KUKA KRL program: MyProgram_090().src

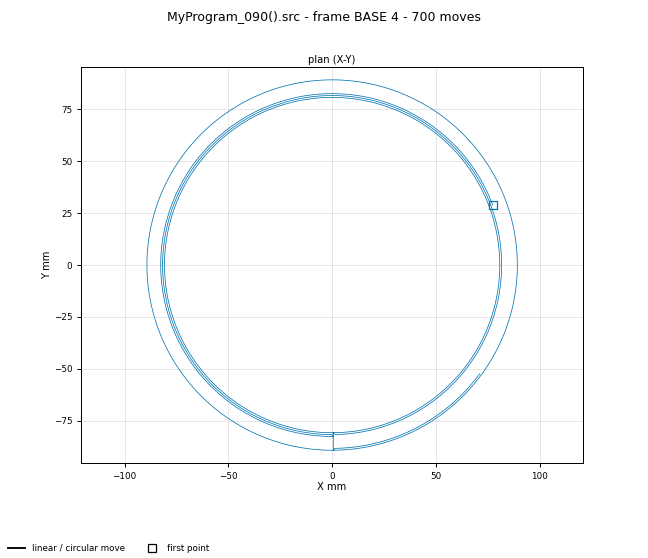
[picture p0: tool path of MyProgram_090().src in frame BASE 4, 700 of 700 moves have a stored position in this frame; points joined in program order, loops and branches not executed]
&ACCESS RVP
&REL 1
&PARAM TEMPLATE = C:\KRC\Roboter\Template\vorgabe
&PARAM EDITMASK = *
DEF MyProgram_090()
; ---- Setting reference (Base) ----
$BASE = BASE_DATA[4]

; --------------------------
; ---- Setting tool (TCP) ----
$TOOL = TOOL_DATA[3]
; --------------------------

$VEL.CP = VEL_APROX_PRINT
Startdeposition()
$VEL.CP = VEL_PRINT
LIN {X 77.3281,Y 28.9448,Z 86,A 15.3349,B 24.9023,C -2.2824,E1 25.1495,E2 429.3591} C_DIS
LIN {X 75.8466,Y 32.631,Z 86,A 18.4549,B 24.9006,C -2.3023,E1 25.1461,E2 426.2095} C_DIS
LIN {X 74.568,Y 35.455,Z 86,A 20.5991,B 24.9001,C -2.3081,E1 25.1436,E2 424.0632} C_DIS
LIN {X 72.599,Y 39.3284,Z 86,A 23.5098,B 24.8996,C -2.3129,E1 25.1398,E2 421.1565} C_DIS
LIN {X 70.8215,Y 42.4488,Z 86,A 26.772,B 24.8968,C -2.3448,E1 25.1351,E2 417.8357} C_DIS
LIN {X 68.6878,Y 45.8205,Z 86,A 28.6373,B 24.8988,C -2.3222,E1 25.1323,E2 416.0329} C_DIS
LIN {X 67.0803,Y 48.1416,Z 86,A 30.6371,B 24.8983,C -2.3285,E1 25.1291,E2 414.0282} C_DIS
LIN {X 63.6188,Y 52.6309,Z 86,A 34.2149,B 24.8985,C -2.3263,E1 25.123,E2 410.4722} C_DIS
LIN {X 61.7276,Y 54.8374,Z 86,A 37.2047,B 24.8953,C -2.3623,E1 25.1174,E2 407.4109} C_DIS
LIN {X 59.4279,Y 57.3206,Z 86,A 39.1109,B 24.8961,C -2.3531,E1 25.1137,E2 405.5347} C_DIS
LIN {X 57.4607,Y 59.2929,Z 86,A 40.8256,B 24.8964,C -2.3501,E1 25.1103,E2 403.8342} C_DIS
LIN {X 55.1536,Y 61.4445,Z 86,A 43.0458,B 24.8959,C -2.3555,E1 25.1058,E2 401.6102} C_DIS
LIN {X 52.6987,Y 63.5625,Z 86,A 45.3521,B 24.8953,C -2.3616,E1 25.1008,E2 399.2985} C_DIS
LIN {X 48.15,Y 67.0743,Z 86,A 49.5371,B 24.8942,C -2.3748,E1 25.0915,E2 395.0973} C_DIS
LIN {X 45.0145,Y 69.219,Z 86,A 51.9336,B 24.8945,C -2.3714,E1 25.0859,E2 392.7168} C_DIS
LIN {X 39.6414,Y 72.4292,Z 86,A 55.9168,B 24.8949,C -2.3664,E1 25.0764,E2 388.7575} C_DIS
LIN {X 35.4802,Y 74.5559,Z 86,A 59.3138,B 24.8941,C -2.3753,E1 25.0679,E2 385.3489} C_DIS
LIN {X 32.5804,Y 75.8687,Z 86,A 61.5876,B 24.8937,C -2.3797,E1 25.0621,E2 383.0701} C_DIS
LIN {X 30.2189,Y 76.8385,Z 86,A 63.6936,B 24.8926,C -2.3918,E1 25.0565,E2 380.9401} C_DIS
LIN {X 26.6751,Y 78.14,Z 86,A 66.6036,B 24.8916,C -2.403,E1 25.0488,E2 378.0094} C_DIS
LIN {X 23.5557,Y 79.1357,Z 86,A 67.8541,B 24.8943,C -2.3735,E1 25.0457,E2 376.8311} C_DIS
LIN {X 20.2883,Y 80.0362,Z 86,A 70.6318,B 24.893,C -2.3879,E1 25.0381,E2 374.0238} C_DIS
LIN {X 17.3744,Y 80.7187,Z 86,A 72.792,B 24.8927,C -2.3915,E1 25.0322,E2 371.858} C_DIS
LIN {X 14.1692,Y 81.3435,Z 86,A 75.1053,B 24.8925,C -2.3937,E1 25.0258,E2 369.5418} C_DIS
LIN {X 11.6124,Y 81.7465,Z 86,A 77.0151,B 24.8921,C -2.3976,E1 25.0205,E2 367.6245} C_DIS
LIN {X 8.7977,Y 82.0973,Z 86,A 78.7957,B 24.8926,C -2.3923,E1 25.0156,E2 365.8578} C_DIS
LIN {X 5.8329,Y 82.3613,Z 86,A 80.8527,B 24.8926,C -2.3922,E1 25.0099,E2 363.8021} C_DIS
LIN {X 2.46,Y 82.5305,Z 86,A 83.3881,B 24.8921,C -2.3977,E1 25.0028,E2 361.2543} C_DIS
LIN {X -1.694,Y 82.5499,Z 86,A 85.9176,B 24.8931,C -2.3867,E1 24.9958,E2 358.751} C_DIS
LIN {X -4.2402,Y 82.4588,Z 86,A 87.9133,B 24.8926,C -2.3927,E1 24.9902,E2 356.7404} C_DIS
LIN {X -7.701,Y 82.2073,Z 86,A 90.4483,B 24.8923,C -2.3954,E1 24.9831,E2 354.198} C_DIS
LIN {X -11.3944,Y 81.7774,Z 86,A 92.4535,B 24.894,C -2.3771,E1 24.9777,E2 352.2347} C_DIS
LIN {X -13.5496,Y 81.4478,Z 86,A 94.2689,B 24.8933,C -2.3848,E1 24.9726,E2 350.3994} C_DIS
LIN {X -16.7265,Y 80.8552,Z 86,A 97.0733,B 24.892,C -2.3992,E1 24.9649,E2 347.5575} C_DIS
LIN {X -20.9138,Y 79.8754,Z 86,A 100.2073,B 24.8918,C -2.4006,E1 24.9564,E2 344.4156} C_DIS
LIN {X -24.2643,Y 78.9213,Z 86,A 102.3651,B 24.8928,C -2.3905,E1 24.9506,E2 342.2784} C_DIS
LIN {X -27.4735,Y 77.8624,Z 86,A 105.2276,B 24.8917,C -2.4024,E1 24.943,E2 339.3818} C_DIS
LIN {X -31.5003,Y 76.3231,Z 86,A 107.3625,B 24.8943,C -2.3738,E1 24.9377,E2 337.3103} C_DIS
LIN {X -34.3091,Y 75.1026,Z 86,A 109.4716,B 24.8946,C -2.3702,E1 24.9323,E2 335.2046} C_DIS
LIN {X -37.1656,Y 73.731,Z 86,A 112.4576,B 24.8929,C -2.3889,E1 24.9247,E2 332.1661} C_DIS
LIN {X -40.6338,Y 71.8778,Z 86,A 114.2221,B 24.8957,C -2.3572,E1 24.9206,E2 330.4722} C_DIS
LIN {X -43.0737,Y 70.4418,Z 86,A 116.6537,B 24.8949,C -2.3666,E1 24.9147,E2 328.0106} C_DIS
LIN {X -46.8346,Y 67.9989,Z 86,A 119.7688,B 24.8954,C -2.3607,E1 24.9075,E2 324.8994} C_DIS
LIN {X -49.3306,Y 66.2113,Z 86,A 121.5161,B 24.8968,C -2.3457,E1 24.9036,E2 323.1816} C_DIS
LIN {X -51.6187,Y 64.4443,Z 86,A 123.7673,B 24.8965,C -2.3482,E1 24.8986,E2 320.9162} C_DIS
LIN {X -53.4699,Y 62.9151,Z 86,A 125.3426,B 24.8971,C -2.342,E1 24.8953,E2 319.3495} C_DIS
LIN {X -55.9727,Y 60.6995,Z 86,A 127.7309,B 24.8974,C -2.3386,E1 24.8903,E2 316.9597} C_DIS
LIN {X -58.3701,Y 58.3994,Z 86,A 130.1929,B 24.8974,C -2.3374,E1 24.8854,E2 314.4903} C_DIS
LIN {X -60.9993,Y 55.646,Z 86,A 132.5499,B 24.8987,C -2.3232,E1 24.881,E2 312.157} C_DIS
LIN {X -63.0145,Y 53.3532,Z 86,A 134.8528,B 24.8987,C -2.3228,E1 24.8767,E2 309.8445} C_DIS
LIN {X -65.1441,Y 50.7324,Z 86,A 137.6368,B 24.8983,C -2.3286,E1 24.8719,E2 307.0336} C_DIS
LIN {X -68.1053,Y 46.6821,Z 86,A 140.6854,B 24.9001,C -2.3074,E1 24.867,E2 304.0206} C_DIS
LIN {X -70.4763,Y 43.0168,Z 86,A 143.9951,B 24.9001,C -2.3064,E1 24.8621,E2 300.6963} C_DIS
LIN {X -72.2097,Y 40.0393,Z 86,A 146.2197,B 24.9012,C -2.2951,E1 24.859,E2 298.4871} C_DIS
LIN {X -74.9102,Y 34.7247,Z 86,A 150.4078,B 24.9021,C -2.2842,E1 24.8539,E2 294.3024} C_DIS
LIN {X -75.9626,Y 32.3591,Z 86,A 152.1687,B 24.9027,C -2.2779,E1 24.8519,E2 292.547} C_DIS
LIN {X -77.3859,Y 28.792,Z 86,A 155.1139,B 24.9027,C -2.2772,E1 24.849,E2 289.5867} C_DIS
LIN {X -78.3928,Y 25.9256,Z 86,A 156.9348,B 24.9039,C -2.263,E1 24.8474,E2 287.7893} C_DIS
LIN {X -79.896,Y 20.8338,Z 86,A 160.5723,B 24.905,C -2.2503,E1 24.8446,E2 284.1612} C_DIS
LIN {X -80.5932,Y 17.9499,Z 86,A 162.7179,B 24.9054,C -2.2461,E1 24.8433,E2 282.0131} C_DIS
LIN {X -81.3182,Y 14.3103,Z 86,A 166.0647,B 24.9043,C -2.2586,E1 24.8416,E2 278.6166} C_DIS
LIN {X -81.9179,Y 10.3374,Z 86,A 168.0108,B 24.907,C -2.2272,E1 24.8409,E2 276.7338} C_DIS
LIN {X -82.1781,Y 8.0167,Z 86,A 169.7244,B 24.9072,C -2.2245,E1 24.8404,E2 275.0165} C_DIS
LIN {X -82.4608,Y 4.2037,Z 86,A 172.2617,B 24.9081,C -2.2129,E1 24.8399,E2 272.4915} C_DIS
LIN {X -82.5537,Y 1.4888,Z 86,A 174.2134,B 24.9085,C -2.2087,E1 24.8398,E2 270.5382} C_DIS
LIN {X -82.5438,Y -2.0277,Z 86,A 176.555,B 24.9094,C -2.1983,E1 24.8398,E2 268.2073} C_DIS
LIN {X -82.4146,Y -5.0392,Z 86,A 178.8476,B 24.9094,C -2.197,E1 24.8402,E2 265.904} C_DIS
LIN {X -82.1848,Y -7.9446,Z 86,A -178.3575,B 24.9083,C -2.2113,E1 24.841,E2 263.0581} C_DIS
LIN {X -81.7181,Y -11.8118,Z 86,A -176.4955,B 24.9108,C -2.1803,E1 24.8416,E2 261.2591} C_DIS
LIN {X -80.6837,Y -17.5348,Z 86,A -172.3512,B 24.9116,C -2.1706,E1 24.8438,E2 257.1132} C_DIS
LIN {X -79.8963,Y -20.8325,Z 86,A -170.024,B 24.9123,C -2.1628,E1 24.8454,E2 254.7912} C_DIS
LIN {X -79.3316,Y -22.8909,Z 86,A -167.3362,B 24.91,C -2.191,E1 24.8476,E2 252.0204} C_DIS
LIN {X -77.7775,Y -27.7156,Z 86,A -164.7586,B 24.9129,C -2.1551,E1 24.8498,E2 249.514} C_DIS
LIN {X -76.5697,Y -30.8945,Z 86,A -162.5845,B 24.9138,C -2.1432,E1 24.852,E2 247.3559} C_DIS
LIN {X -75.4207,Y -33.6031,Z 86,A -160.5049,B 24.9142,C -2.1385,E1 24.8544,E2 245.2763} C_DIS
LIN {X -74.1285,Y -36.365,Z 86,A -158.3588,B 24.9146,C -2.1334,E1 24.857,E2 243.1307} C_DIS
LIN {X -72.0249,Y -40.3702,Z 86,A -155.0625,B 24.915,C -2.1292,E1 24.8613,E2 239.8269} C_DIS
LIN {X -69.3806,Y -44.7627,Z 86,A -151.6258,B 24.916,C -2.1166,E1 24.8664,E2 236.4027} C_DIS
LIN {X -67.4996,Y -47.554,Z 86,A -148.4036,B 24.9145,C -2.1353,E1 24.8716,E2 233.1201} C_DIS
LIN {X -64.8603,Y -51.0929,Z 86,A -146.635,B 24.9179,C -2.0922,E1 24.8745,E2 231.4459} C_DIS
LIN {X -62.2386,Y -54.2559,Z 86,A -142.7938,B 24.9163,C -2.113,E1 24.8815,E2 227.5374} C_DIS
LIN {X -60.0446,Y -56.6746,Z 86,A -141.2475,B 24.9182,C -2.088,E1 24.8844,E2 226.044} C_DIS
LIN {X -58.2822,Y -58.4863,Z 86,A -139.2971,B 24.9182,C -2.0898,E1 24.8882,E2 224.0811} C_DIS
LIN {X -54.727,Y -61.8264,Z 86,A -136.136,B 24.9191,C -2.0767,E1 24.8947,E2 220.9383} C_DIS
LIN {X -51.2494,Y -64.7367,Z 86,A -132.4233,B 24.9183,C -2.0868,E1 24.9028,E2 217.1874} C_DIS
LIN {X -47.5417,Y -67.5083,Z 86,A -129.4906,B 24.9194,C -2.0734,E1 24.9093,E2 214.2764} C_DIS
LIN {X -45.2055,Y -69.0932,Z 86,A -127.0426,B 24.9185,C -2.0844,E1 24.9151,E2 211.7943} C_DIS
LIN {X -41.413,Y -71.431,Z 86,A -124.0005,B 24.919,C -2.0785,E1 24.9224,E2 208.7569} C_DIS
LIN {X -37.1468,Y -73.7406,Z 86,A -120.9339,B 24.92,C -2.0655,E1 24.93,E2 205.7128} C_DIS
LIN {X -34.1894,Y -75.1565,Z 86,A -118.8468,B 24.9206,C -2.0575,E1 24.9352,E2 203.6396} C_DIS
LIN {X -30.8787,Y -76.5762,Z 86,A -116.3984,B 24.9209,C -2.0534,E1 24.9415,E2 201.1952} C_DIS
LIN {X -26.6206,Y -78.1584,Z 86,A -113.4742,B 24.9217,C -2.044,E1 24.9492,E2 198.2876} C_DIS
LIN {X -24.1171,Y -78.9672,Z 86,A -111.2313,B 24.9208,C -2.0549,E1 24.9552,E2 196.0149} C_DIS
LIN {X -20.8123,Y -79.9015,Z 86,A -108.9288,B 24.9211,C -2.051,E1 24.9614,E2 193.718} C_DIS
LIN {X -17.7972,Y -80.6265,Z 86,A -106.6486,B 24.9209,C -2.0538,E1 24.9676,E2 191.4283} C_DIS
LIN {X -14.6611,Y -81.2551,Z 86,A -104.2027,B 24.9204,C -2.0597,E1 24.9744,E2 188.9656} C_DIS
LIN {X -10.524,Y -81.8937,Z 86,A -101.6715,B 24.9214,C -2.0479,E1 24.9813,E2 186.4605} C_DIS
LIN {X -7.454,Y -82.2301,Z 86,A -99.5955,B 24.9215,C -2.0457,E1 24.9871,E2 184.3887} C_DIS
LIN {X -3.4693,Y -82.4943,Z 86,A -96.4906,B 24.9207,C -2.0559,E1 24.9958,E2 181.2585} C_DIS
LIN {X 0.5302,Y -82.5625,Z 86,A -94.6776,B 24.9229,C -2.0274,E1 25.0007,E2 179.5132} C_DIS
Enddeposition()
LIN {X 0.5302,Y -82.5625,Z 86,A -94.6776,B 24.9229,C -2.0274,E1 25.0007,E2 179.5132} C_DIS
Startdeposition()
$VEL.CP = VEL_PRINT
LIN {X -0.0163,Y -81.6615,Z 86,A -95.4197,B 24.9225,C -2.0324,E1 24.9986,E2 180.2432} C_DIS
LIN {X -2.7317,Y -81.6147,Z 86,A -97.1926,B 24.9223,C -2.0361,E1 24.9937,E2 182.0077} C_DIS
LIN {X -5.5212,Y -81.4732,Z 86,A -99.1546,B 24.9223,C -2.0359,E1 24.9882,E2 183.9707} C_DIS
LIN {X -8.4748,Y -81.2191,Z 86,A -101.2543,B 24.9223,C -2.0355,E1 24.9824,E2 186.0724} C_DIS
LIN {X -11.4403,Y -80.8547,Z 86,A -103.348,B 24.9223,C -2.036,E1 24.9766,E2 188.1666} C_DIS
LIN {X -14.2538,Y -80.4067,Z 86,A -105.405,B 24.9223,C -2.0349,E1 24.9709,E2 190.2281} C_DIS
LIN {X -17.4514,Y -79.7735,Z 86,A -107.7669,B 24.9224,C -2.0337,E1 24.9644,E2 192.5956} C_DIS
LIN {X -20.8127,Y -78.9648,Z 86,A -110.2307,B 24.9224,C -2.034,E1 24.9578,E2 195.0624} C_DIS
LIN {X -24.2019,Y -77.9912,Z 86,A -112.6185,B 24.9221,C -2.0382,E1 24.9514,E2 197.4442} C_DIS
LIN {X -27.44,Y -76.9129,Z 86,A -115.1204,B 24.9221,C -2.0371,E1 24.9448,E2 199.9535} C_DIS
LIN {X -30.5238,Y -75.7413,Z 86,A -117.3329,B 24.9218,C -2.0422,E1 24.939,E2 202.1586} C_DIS
LIN {X -33.4971,Y -74.4736,Z 86,A -119.5845,B 24.9216,C -2.0451,E1 24.9333,E2 204.4086} C_DIS
LIN {X -36.4481,Y -73.0749,Z 86,A -121.9228,B 24.9215,C -2.0465,E1 24.9274,E2 206.7497} C_DIS
LIN {X -39.2907,Y -71.5875,Z 86,A -124.3132,B 24.9215,C -2.0455,E1 24.9215,E2 209.149} C_DIS
LIN {X -41.5941,Y -70.273,Z 86,A -126.0513,B 24.9211,C -2.0516,E1 24.9173,E2 210.878} C_DIS
LIN {X -44.204,Y -68.6613,Z 86,A -128.0921,B 24.9206,C -2.0579,E1 24.9125,E2 212.9102} C_DIS
LIN {X -46.6315,Y -67.0363,Z 86,A -130.1603,B 24.9204,C -2.0607,E1 24.9077,E2 214.9787} C_DIS
LIN {X -49.0247,Y -65.3066,Z 86,A -133.1291,B 24.922,C -2.0399,E1 24.901,E2 218.0076} C_DIS
LIN {X -52.1622,Y -62.8289,Z 86,A -135.0796,B 24.9198,C -2.0681,E1 24.8969,E2 219.8982} C_DIS
LIN {X -54.3609,Y -60.9367,Z 86,A -137.5367,B 24.9204,C -2.0607,E1 24.8917,E2 222.3827} C_DIS
LIN {X -57.3481,Y -58.134,Z 86,A -140.1183,B 24.9193,C -2.0744,E1 24.8865,E2 224.9423} C_DIS
LIN {X -59.4283,Y -56.0058,Z 86,A -142.8327,B 24.9203,C -2.0622,E1 24.8812,E2 227.6976} C_DIS
LIN {X -61.8542,Y -53.3164,Z 86,A -144.7929,B 24.9186,C -2.0834,E1 24.8777,E2 229.6163} C_DIS
LIN {X -64.183,Y -50.487,Z 86,A -147.1554,B 24.9177,C -2.095,E1 24.8736,E2 231.9621} C_DIS
LIN {X -66.2039,Y -47.8082,Z 86,A -149.7166,B 24.9177,C -2.0952,E1 24.8693,E2 234.5351} C_DIS
LIN {X -68.0014,Y -45.2136,Z 86,A -151.9136,B 24.9172,C -2.1012,E1 24.8659,E2 236.7287} C_DIS
LIN {X -69.6279,Y -42.6663,Z 86,A -154.3798,B 24.9175,C -2.0976,E1 24.8622,E2 239.2161} C_DIS
LIN {X -72.238,Y -38.0794,Z 86,A -157.7911,B 24.9161,C -2.1152,E1 24.8576,E2 242.6033} C_DIS
LIN {X -73.688,Y -35.192,Z 86,A -160.1175,B 24.9157,C -2.1199,E1 24.8548,E2 244.931} C_DIS
LIN {X -75.1122,Y -32.0414,Z 86,A -162.5168,B 24.9151,C -2.1275,E1 24.8521,E2 247.3255} C_DIS
LIN {X -76.3612,Y -28.9367,Z 86,A -164.8125,B 24.9145,C -2.1357,E1 24.8497,E2 249.6145} C_DIS
LIN {X -77.739,Y -25.0006,Z 86,A -167.7777,B 24.9138,C -2.1433,E1 24.8471,E2 252.5785} C_DIS
LIN {X -78.6619,Y -21.927,Z 86,A -169.7895,B 24.9128,C -2.1562,E1 24.8455,E2 254.571} C_DIS
LIN {X -79.5463,Y -18.4598,Z 86,A -172.518,B 24.9126,C -2.1582,E1 24.8437,E2 257.3107} C_DIS
LIN {X -80.6981,Y -12.4973,Z 86,A -177.8758,B 24.9138,C -2.1435,E1 24.8411,E2 262.7355} C_DIS
LIN {X -81.2753,Y -7.9295,Z 86,A 179.9404,B 24.9108,C -2.1802,E1 24.8404,E2 264.8446} C_DIS
LIN {X -81.4834,Y -5.3695,Z 86,A 178.0036,B 24.9107,C -2.1825,E1 24.84,E2 266.7876} C_DIS
LIN {X -81.6368,Y -2.0114,Z 86,A 175.5316,B 24.9103,C -2.1871,E1 24.8398,E2 269.2636} C_DIS
LIN {X -81.6507,Y 1.2603,Z 86,A 173.367,B 24.9094,C -2.1977,E1 24.8398,E2 271.4157} C_DIS
LIN {X -81.5318,Y 4.5754,Z 86,A 170.3679,B 24.9102,C -2.1881,E1 24.8403,E2 274.4559} C_DIS
LIN {X -81.2554,Y 8.1284,Z 86,A 168.4292,B 24.9084,C -2.2103,E1 24.8408,E2 276.3532} C_DIS
LIN {X -80.6413,Y 12.8647,Z 86,A 165.1268,B 24.9074,C -2.2222,E1 24.842,E2 279.6469} C_DIS
LIN {X -80.1601,Y 15.5802,Z 86,A 163.3021,B 24.9066,C -2.2312,E1 24.843,E2 281.4609} C_DIS
LIN {X -79.4501,Y 18.8757,Z 86,A 160.6417,B 24.9066,C -2.2311,E1 24.8446,E2 284.1373} C_DIS
LIN {X -78.6107,Y 22.1078,Z 86,A 158.3187,B 24.906,C -2.239,E1 24.8463,E2 286.455} C_DIS
LIN {X -77.6206,Y 25.3667,Z 86,A 156.0491,B 24.9051,C -2.2494,E1 24.8482,E2 288.7125} C_DIS
LIN {X -76.7091,Y 28.0015,Z 86,A 154.0454,B 24.9047,C -2.2542,E1 24.8501,E2 290.7162} C_DIS
LIN {X -75.5189,Y 31.0701,Z 86,A 151.6412,B 24.9043,C -2.2588,E1 24.8526,E2 293.123} C_DIS
LIN {X -74.1724,Y 34.1603,Z 86,A 148.6165,B 24.9051,C -2.249,E1 24.8561,E2 296.1876} C_DIS
LIN {X -72.4982,Y 37.5844,Z 86,A 146.5396,B 24.9032,C -2.2721,E1 24.8587,E2 298.2205} C_DIS
LIN {X -70.7317,Y 40.8094,Z 86,A 143.0615,B 24.9045,C -2.2565,E1 24.8636,E2 301.7538} C_DIS
LIN {X -68.3228,Y 44.7262,Z 86,A 140.8,B 24.9016,C -2.2903,E1 24.8669,E2 303.9462} C_DIS
LIN {X -66.4126,Y 47.5157,Z 86,A 138.6725,B 24.9005,C -2.3031,E1 24.8703,E2 306.0536} C_DIS
LIN {X -64.9897,Y 49.4465,Z 86,A 136.6632,B 24.9008,C -2.2991,E1 24.8737,E2 308.0822} C_DIS
LIN {X -62.9326,Y 52.0374,Z 86,A 134.4024,B 24.9002,C -2.3067,E1 24.8776,E2 310.3353} C_DIS
LIN {X -60.745,Y 54.575,Z 86,A 132.1796,B 24.8994,C -2.316,E1 24.8817,E2 312.5459} C_DIS
LIN {X -58.701,Y 56.7677,Z 86,A 129.9101,B 24.8993,C -2.3168,E1 24.8861,E2 314.8235} C_DIS
LIN {X -56.3794,Y 59.0753,Z 86,A 127.5483,B 24.899,C -2.3205,E1 24.8908,E2 317.1863} C_DIS
LIN {X -53.9154,Y 61.3316,Z 86,A 125.2446,B 24.8984,C -2.3269,E1 24.8956,E2 319.4839} C_DIS
LIN {X -51.7238,Y 63.1915,Z 86,A 123.186,B 24.8981,C -2.3302,E1 24.9,E2 321.5425} C_DIS
LIN {X -49.1123,Y 65.2407,Z 86,A 121.1232,B 24.8971,C -2.3422,E1 24.9045,E2 323.5842} C_DIS
LIN {X -47.4404,Y 66.4663,Z 86,A 118.8847,B 24.8986,C -2.3243,E1 24.9097,E2 325.8732} C_DIS
LIN {X -44.7816,Y 68.2863,Z 86,A 116.454,B 24.8986,C -2.3241,E1 24.9154,E2 328.3123} C_DIS
LIN {X -41.653,Y 70.2382,Z 86,A 114.7603,B 24.8961,C -2.3527,E1 24.9193,E2 329.9431} C_DIS
LIN {X -39.637,Y 71.3952,Z 86,A 112.837,B 24.8966,C -2.3476,E1 24.924,E2 331.884} C_DIS
LIN {X -36.8015,Y 72.8984,Z 86,A 110.6742,B 24.8961,C -2.3537,E1 24.9294,E2 334.0383} C_DIS
LIN {X -34.1579,Y 74.1736,Z 86,A 108.5988,B 24.8958,C -2.3564,E1 24.9346,E2 336.1125} C_DIS
LIN {X -31.4321,Y 75.369,Z 86,A 106.7351,B 24.895,C -2.3656,E1 24.9393,E2 337.9587} C_DIS
LIN {X -28.6976,Y 76.4517,Z 86,A 104.3917,B 24.8954,C -2.3606,E1 24.9455,E2 340.3189} C_DIS
LIN {X -21.8708,Y 78.6778,Z 86,A 99.3214,B 24.895,C -2.3655,E1 24.959,E2 345.3865} C_DIS
LIN {X -19.5564,Y 79.284,Z 86,A 97.2603,B 24.8958,C -2.3565,E1 24.9646,E2 347.4719} C_DIS
LIN {X -15.3506,Y 80.2043,Z 86,A 94.6229,B 24.8946,C -2.3697,E1 24.9718,E2 350.081} C_DIS
LIN {X -11.9533,Y 80.7818,Z 86,A 92.2046,B 24.8945,C -2.3713,E1 24.9784,E2 352.4976} C_DIS
LIN {X -8.6247,Y 81.2034,Z 86,A 89.9178,B 24.8942,C -2.3746,E1 24.9847,E2 354.7782} C_DIS
LIN {X -5.3735,Y 81.4832,Z 86,A 87.5849,B 24.8942,C -2.3744,E1 24.9912,E2 357.1126} C_DIS
LIN {X -2.1477,Y 81.6326,Z 86,A 85.2523,B 24.8943,C -2.3731,E1 24.9978,E2 359.4485} C_DIS
LIN {X 0.7959,Y 81.6567,Z 86,A 83.2701,B 24.8941,C -2.3759,E1 25.0033,E2 361.4241} C_DIS
LIN {X 3.8268,Y 81.571,Z 86,A 81.1152,B 24.8941,C -2.3753,E1 25.0093,E2 363.5799} C_DIS
LIN {X 7.0016,Y 81.3608,Z 86,A 78.8568,B 24.8942,C -2.3744,E1 25.0156,E2 365.8392} C_DIS
LIN {X 10.1009,Y 81.0339,Z 86,A 76.5967,B 24.8944,C -2.3719,E1 25.0219,E2 368.1036} C_DIS
LIN {X 13.674,Y 80.5073,Z 86,A 74.1306,B 24.8944,C -2.3731,E1 25.0287,E2 370.5644} C_DIS
LIN {X 17.0505,Y 79.861,Z 86,A 71.7533,B 24.8944,C -2.3731,E1 25.0352,E2 372.9389} C_DIS
LIN {X 20.3019,Y 79.0961,Z 86,A 69.3962,B 24.8944,C -2.3714,E1 25.0415,E2 375.2967} C_DIS
LIN {X 22.6908,Y 78.4455,Z 86,A 67.5493,B 24.8949,C -2.3669,E1 25.0465,E2 377.151} C_DIS
LIN {X 26.3137,Y 77.3047,Z 86,A 65.1603,B 24.8943,C -2.373,E1 25.0528,E2 379.5211} C_DIS
LIN {X 29.1854,Y 76.267,Z 86,A 62.8576,B 24.8949,C -2.3662,E1 25.0589,E2 381.835} C_DIS
LIN {X 32.1987,Y 75.0456,Z 86,A 60.5629,B 24.8952,C -2.3634,E1 25.0648,E2 384.131} C_DIS
LIN {X 35.1906,Y 73.6887,Z 86,A 58.6446,B 24.8944,C -2.3724,E1 25.0696,E2 386.023} C_DIS
LIN {X 37.1119,Y 72.7398,Z 86,A 56.8295,B 24.8954,C -2.3611,E1 25.0742,E2 387.86} C_DIS
LIN {X 41.0462,Y 70.5957,Z 86,A 53.6999,B 24.8957,C -2.3572,E1 25.0818,E2 390.9897} C_DIS
LIN {X 43.7179,Y 68.9734,Z 86,A 51.3663,B 24.8964,C -2.3496,E1 25.0874,E2 393.3339} C_DIS
LIN {X 46.4722,Y 67.147,Z 86,A 48.328,B 24.8987,C -2.324,E1 25.0945,E2 396.4225} C_DIS
LIN {X 49.8708,Y 64.6627,Z 86,A 46.1209,B 24.8971,C -2.3415,E1 25.0993,E2 398.5802} C_DIS
LIN {X 52.7098,Y 62.3711,Z 86,A 43.7813,B 24.897,C -2.3435,E1 25.1043,E2 400.9062} C_DIS
LIN {X 54.9109,Y 60.4427,Z 86,A 41.6015,B 24.8977,C -2.3355,E1 25.1088,E2 403.0961} C_DIS
LIN {X 57.358,Y 58.1242,Z 86,A 39.472,B 24.8974,C -2.3379,E1 25.1131,E2 405.2109} C_DIS
LIN {X 60.0163,Y 55.3756,Z 86,A 36.2499,B 24.8994,C -2.3153,E1 25.1194,E2 408.4726} C_DIS
LIN {X 62.6228,Y 52.4102,Z 86,A 33.8338,B 24.899,C -2.32,E1 25.1237,E2 410.8666} C_DIS
LIN {X 64.7591,Y 49.7458,Z 86,A 31.5207,B 24.8993,C -2.3169,E1 25.1277,E2 413.1762} C_DIS
LIN {X 66.531,Y 47.3498,Z 86,A 29.3373,B 24.9,C -2.3088,E1 25.1313,E2 415.3681} C_DIS
LIN {X 68.29,Y 44.7759,Z 86,A 27.3863,B 24.8998,C -2.3108,E1 25.1343,E2 417.3048} C_DIS
LIN {X 70.0435,Y 41.9824,Z 86,A 24.8252,B 24.901,C -2.2969,E1 25.1381,E2 419.8857} C_DIS
LIN {X 71.638,Y 39.1976,Z 86,A 22.6358,B 24.9014,C -2.2928,E1 25.141,E2 422.0734} C_DIS
LIN {X 73.2188,Y 36.1579,Z 86,A 20.2943,B 24.9018,C -2.2882,E1 25.144,E2 424.4133} C_DIS
LIN {X 74.6029,Y 33.21,Z 86,A 18.0169,B 24.9023,C -2.282,E1 25.1466,E2 426.693} C_DIS
LIN {X 75.8489,Y 30.2572,Z 86,A 15.7488,B 24.9029,C -2.2749,E1 25.1491,E2 428.9653} C_DIS
LIN {X 77.1515,Y 26.7601,Z 86,A 12.9736,B 24.904,C -2.2622,E1 25.1517,E2 431.755} C_DIS
LIN {X 78.3549,Y 22.9985,Z 86,A 10.4431,B 24.904,C -2.2616,E1 25.1538,E2 434.2723} C_DIS
LIN {X 79.2223,Y 19.8095,Z 86,A 8.0579,B 24.9048,C -2.2525,E1 25.1554,E2 436.6656} C_DIS
LIN {X 79.9948,Y 16.4073,Z 86,A 5.7311,B 24.9051,C -2.2489,E1 25.1568,E2 438.9874} C_DIS
LIN {X 80.4429,Y 14.0526,Z 86,A 4.0452,B 24.9056,C -2.2435,E1 25.1577,E2 440.676} C_DIS
LIN {X 80.8968,Y 11.1438,Z 86,A 1.993,B 24.9061,C -2.2375,E1 25.1585,E2 442.7303} C_DIS
LIN {X 81.2503,Y 8.177,Z 86,A -0.1945,B 24.9069,C -2.2279,E1 25.1592,E2 444.9275} C_DIS
LIN {X 81.5224,Y 4.7449,Z 86,A -2.5734,B 24.9074,C -2.2214,E1 25.1596,E2 447.3075} C_DIS
LIN {X 81.6487,Y 1.3656,Z 86,A -4.8641,B 24.9078,C -2.2165,E1 25.1598,E2 449.5961} C_DIS
LIN {X 81.6554,Y -1.0033,Z 86,A -6.5354,B 24.9083,C -2.2109,E1 25.1598,E2 451.2708} C_DIS
LIN {X 81.5592,Y -4.0789,Z 86,A -8.7254,B 24.909,C -2.203,E1 25.1595,E2 453.4665} C_DIS
LIN {X 81.3102,Y -7.5512,Z 86,A -11.0689,B 24.9093,C -2.1984,E1 25.159,E2 455.8069} C_DIS
LIN {X 81.0403,Y -10.0514,Z 86,A -12.8729,B 24.9099,C -2.1915,E1 25.1584,E2 457.6166} C_DIS
LIN {X 80.5587,Y -13.3667,Z 86,A -15.1415,B 24.9103,C -2.1866,E1 25.1574,E2 459.8833} C_DIS
LIN {X 79.9493,Y -16.6289,Z 86,A -17.407,B 24.9108,C -2.1813,E1 25.1562,E2 462.1481} C_DIS
LIN {X 79.3715,Y -19.1979,Z 86,A -20.5564,B 24.9146,C -2.1337,E1 25.154,E2 465.3918} C_DIS
LIN {X 77.9181,Y -24.4378,Z 86,A -22.9943,B 24.912,C -2.1659,E1 25.1521,E2 467.7396} C_DIS
LIN {X 76.7657,Y -27.8463,Z 86,A -25.5583,B 24.9127,C -2.1568,E1 25.1498,E2 470.3106} C_DIS
LIN {X 75.6172,Y -30.8285,Z 86,A -27.7867,B 24.9133,C -2.1505,E1 25.1475,E2 472.5417} C_DIS
LIN {X 74.8075,Y -32.7448,Z 86,A -29.4653,B 24.9142,C -2.139,E1 25.1456,E2 474.2383} C_DIS
LIN {X 73.261,Y -36.0727,Z 86,A -31.8448,B 24.9143,C -2.1376,E1 25.1427,E2 476.6083} C_DIS
LIN {X 71.7012,Y -39.081,Z 86,A -34.2357,B 24.9149,C -2.1302,E1 25.1396,E2 479.004} C_DIS
LIN {X 70.2881,Y -41.5686,Z 86,A -36.1129,B 24.915,C -2.1286,E1 25.137,E2 480.8752} C_DIS
LIN {X 68.6862,Y -44.1653,Z 86,A -38.3023,B 24.9156,C -2.121,E1 25.1337,E2 483.0715} C_DIS
LIN {X 66.9188,Y -46.8005,Z 86,A -40.285,B 24.9155,C -2.1227,E1 25.1306,E2 485.0405} C_DIS
LIN {X 65.754,Y -48.4234,Z 86,A -42.0504,B 24.9167,C -2.1072,E1 25.1277,E2 486.834} C_DIS
LIN {X 63.6009,Y -51.2187,Z 86,A -44.3963,B 24.9169,C -2.1048,E1 25.1236,E2 489.1745} C_DIS
LIN {X 61.4242,Y -53.8093,Z 86,A -46.7862,B 24.9174,C -2.0982,E1 25.1193,E2 491.5692} C_DIS
LIN {X 59.1146,Y -56.338,Z 86,A -49.3452,B 24.9183,C -2.0873,E1 25.1144,E2 494.1428} C_DIS
LIN {X 56.4681,Y -58.9898,Z 86,A -51.7894,B 24.9183,C -2.0868,E1 25.1095,E2 496.5779} C_DIS
LIN {X 54.0073,Y -61.2513,Z 86,A -54.1353,B 24.9188,C -2.0814,E1 25.1046,E2 498.9272} C_DIS
LIN {X 51.2678,Y -63.5611,Z 86,A -56.557,B 24.919,C -2.0787,E1 25.0994,E2 501.3459} C_DIS
LIN {X 48.8961,Y -65.4031,Z 86,A -58.5284,B 24.919,C -2.0785,E1 25.0951,E2 503.3106} C_DIS
LIN {X 46.7139,Y -66.9791,Z 86,A -60.5263,B 24.9195,C -2.0713,E1 25.0905,E2 505.3188} C_DIS
LIN {X 44.128,Y -68.7101,Z 86,A -62.6747,B 24.9198,C -2.0681,E1 25.0855,E2 507.4675} C_DIS
LIN {X 41.1976,Y -70.5074,Z 86,A -65.191,B 24.9204,C -2.0604,E1 25.0794,E2 509.9942} C_DIS
LIN {X 38.3028,Y -72.1203,Z 86,A -67.2891,B 24.9202,C -2.0635,E1 25.0743,E2 512.079} C_DIS
LIN {X 34.1381,Y -74.1827,Z 86,A -70.6866,B 24.9209,C -2.054,E1 25.0658,E2 515.49} C_DIS
LIN {X 31.3328,Y -75.4108,Z 86,A -72.812,B 24.9211,C -2.0515,E1 25.0603,E2 517.6161} C_DIS
LIN {X 29.1671,Y -76.2739,Z 86,A -74.9374,B 24.9224,C -2.0344,E1 25.0547,E2 519.7776} C_DIS
LIN {X 24.1493,Y -78.0075,Z 86,A -77.6544,B 24.9204,C -2.0606,E1 25.0477,E2 522.4272} C_DIS
LIN {X 20.8205,Y -78.9627,Z 86,A -80.7071,B 24.922,C -2.0389,E1 25.0393,E2 525.5263} C_DIS
LIN {X 17.4182,Y -79.7808,Z 86,A -83.1489,B 24.9222,C -2.037,E1 25.0327,E2 527.9692} C_DIS
LIN {X 13.9777,Y -80.4563,Z 86,A -85.5967,B 24.9223,C -2.0354,E1 25.026,E2 530.4181} C_DIS
LIN {X 10.7153,Y -80.9543,Z 86,A -87.8363,B 24.9223,C -2.0361,E1 25.0198,E2 532.654} C_DIS
LIN {X 7.3678,Y -81.3271,Z 86,A -90.0706,B 24.9221,C -2.0386,E1 25.0136,E2 534.8808} C_DIS
LIN {X 4.529,Y -81.5344,Z 86,A -92.1176,B 24.9222,C -2.0363,E1 25.0079,E2 536.9325} C_DIS
LIN {X 1.5273,Y -81.6458,Z 86,A -94.237,B 24.9223,C -2.0352,E1 25.0019,E2 539.0539} C_DIS
LIN {X 1.5273,Y -81.6458,Z 86,A -94.237,B 24.9223,C -2.0352,E1 25.0019,E2 539.0539} C_DIS
Enddeposition()
LIN {X 0.5155,Y -80.7513,Z 86,A -94.535,B 24.9202,C -2.0631,E1 25.0013,E2 539.2859} C_DIS
Startdeposition()
$VEL.CP = VEL_PRINT
LIN {X 2.9646,Y -80.7,Z 86,A -92.3075,B 24.919,C -2.0781,E1 25.0076,E2 537.0231} C_DIS
LIN {X 5.8866,Y -80.5393,Z 86,A -90.3818,B 24.9193,C -2.0745,E1 25.013,E2 535.1068} C_DIS
LIN {X 8.4611,Y -80.3085,Z 86,A -88.4653,B 24.919,C -2.078,E1 25.0183,E2 533.1832} C_DIS
LIN {X 10.865,Y -80.0202,Z 86,A -86.8347,B 24.9191,C -2.0764,E1 25.0228,E2 531.5576} C_DIS
LIN {X 12.784,Y -79.7359,Z 86,A -85.4603,B 24.9191,C -2.0773,E1 25.0266,E2 530.1824} C_DIS
LIN {X 14.7708,Y -79.3921,Z 86,A -84.0156,B 24.919,C -2.0789,E1 25.0306,E2 528.7355} C_DIS
LIN {X 17.4309,Y -78.8496,Z 86,A -82.074,B 24.9188,C -2.0811,E1 25.0359,E2 526.7912} C_DIS
LIN {X 19.6234,Y -78.334,Z 86,A -80.2738,B 24.9182,C -2.0888,E1 25.0408,E2 524.9754} C_DIS
LIN {X 22.485,Y -77.561,Z 86,A -78.1946,B 24.9181,C -2.0904,E1 25.0464,E2 522.8959} C_DIS
LIN {X 25.2932,Y -76.691,Z 86,A -76.3379,B 24.9184,C -2.0858,E1 25.0513,E2 521.0534} C_DIS
LIN {X 27.1118,Y -76.0667,Z 86,A -74.9817,B 24.9183,C -2.0873,E1 25.0549,E2 519.6964} C_DIS
LIN {X 29.0299,Y -75.356,Z 86,A -73.2739,B 24.9175,C -2.0972,E1 25.0594,E2 517.9689} C_DIS
LIN {X 31.8031,Y -74.2283,Z 86,A -71.4116,B 24.9179,C -2.0921,E1 25.0641,E2 516.1229} C_DIS
LIN {X 33.5235,Y -73.4668,Z 86,A -70.0779,B 24.9178,C -2.0941,E1 25.0675,E2 514.7878} C_DIS
LIN {X 35.3817,Y -72.5905,Z 86,A -68.6285,B 24.9176,C -2.0962,E1 25.0712,E2 513.3373} C_DIS
LIN {X 37.1346,Y -71.7095,Z 86,A -67.0808,B 24.917,C -2.1034,E1 25.0751,E2 511.7769} C_DIS
LIN {X 39.7655,Y -70.2848,Z 86,A -64.9404,B 24.9167,C -2.1076,E1 25.0803,E2 509.6326} C_DIS
LIN {X 42.3373,Y -68.7664,Z 86,A -63.0119,B 24.9169,C -2.1055,E1 25.0849,E2 507.7151} C_DIS
LIN {X 44.0079,Y -67.7093,Z 86,A -61.6196,B 24.9167,C -2.1079,E1 25.0882,E2 506.3217} C_DIS
LIN {X 45.684,Y -66.5902,Z 86,A -60.1957,B 24.9165,C -2.1106,E1 25.0915,E2 504.8963} C_DIS
LIN {X 47.3005,Y -65.4519,Z 86,A -58.7991,B 24.9162,C -2.1132,E1 25.0946,E2 503.4983} C_DIS
LIN {X 49.2814,Y -63.9717,Z 86,A -56.9451,B 24.9157,C -2.1201,E1 25.0988,E2 501.6348} C_DIS
LIN {X 51.616,Y -62.1033,Z 86,A -54.8333,B 24.9154,C -2.1244,E1 25.1034,E2 499.5208} C_DIS
LIN {X 53.8461,Y -60.1801,Z 86,A -52.7495,B 24.915,C -2.129,E1 25.1078,E2 497.4343} C_DIS
LIN {X 56.0319,Y -58.1504,Z 86,A -50.6495,B 24.9146,C -2.1335,E1 25.112,E2 495.3324} C_DIS
LIN {X 58.1269,Y -56.0563,Z 86,A -48.5542,B 24.9142,C -2.1384,E1 25.1161,E2 493.2344} C_DIS
LIN {X 60.154,Y -53.8752,Z 86,A -46.4502,B 24.9138,C -2.1434,E1 25.1201,E2 491.1278} C_DIS
LIN {X 62.1029,Y -51.6166,Z 86,A -44.3509,B 24.9134,C -2.1483,E1 25.1239,E2 489.0265} C_DIS
LIN {X 63.9549,Y -49.3033,Z 86,A -42.265,B 24.913,C -2.1534,E1 25.1275,E2 486.9385} C_DIS
LIN {X 65.7136,Y -46.9336,Z 86,A -40.1713,B 24.9126,C -2.159,E1 25.1309,E2 484.8416} C_DIS
LIN {X 67.1226,Y -44.8977,Z 86,A -38.5416,B 24.9126,C -2.1598,E1 25.1335,E2 483.2181} C_DIS
LIN {X 68.2224,Y -43.2086,Z 86,A -37.119,B 24.9122,C -2.1636,E1 25.1356,E2 481.7937} C_DIS
LIN {X 69.4886,Y -41.1386,Z 86,A -35.2888,B 24.9115,C -2.172,E1 25.1383,E2 479.953} C_DIS
LIN {X 70.7372,Y -38.9553,Z 86,A -33.6357,B 24.9115,C -2.1729,E1 25.1405,E2 478.3064} C_DIS
LIN {X 71.6632,Y -37.2242,Z 86,A -32.2534,B 24.9111,C -2.1766,E1 25.1423,E2 476.9225} C_DIS
LIN {X 72.5538,Y -35.457,Z 86,A -30.8587,B 24.9108,C -2.1805,E1 25.1441,E2 475.5262} C_DIS
LIN {X 73.428,Y -33.6095,Z 86,A -29.4212,B 24.9105,C -2.1844,E1 25.1458,E2 474.0872} C_DIS
LIN {X 74.2265,Y -31.8072,Z 86,A -28.0315,B 24.9102,C -2.1883,E1 25.1473,E2 472.6958} C_DIS
LIN {X 75.2273,Y -29.3587,Z 86,A -26.1147,B 24.9096,C -2.1954,E1 25.1493,E2 470.773} C_DIS
LIN {X 76.0288,Y -27.2195,Z 86,A -24.5544,B 24.9093,C -2.1984,E1 25.1508,E2 469.2144} C_DIS
LIN {X 76.6703,Y -25.3561,Z 86,A -23.1711,B 24.909,C -2.2022,E1 25.1521,E2 467.8298} C_DIS
LIN {X 77.5512,Y -22.5181,Z 86,A -21.072,B 24.9085,C -2.2085,E1 25.1538,E2 465.7278} C_DIS
LIN {X 78.2469,Y -19.9623,Z 86,A -18.9483,B 24.9074,C -2.2224,E1 25.1553,E2 463.5835} C_DIS
LIN {X 79.0057,Y -16.7144,Z 86,A -16.8621,B 24.9074,C -2.2207,E1 25.1565,E2 461.5134} C_DIS
LIN {X 79.3917,Y -14.7727,Z 86,A -15.4661,B 24.9071,C -2.2249,E1 25.1573,E2 460.1157} C_DIS
LIN {X 79.7298,Y -12.8235,Z 86,A -14.0677,B 24.9068,C -2.2292,E1 25.1579,E2 458.7154} C_DIS
LIN {X 80.02,Y -10.8665,Z 86,A -12.4244,B 24.9057,C -2.2415,E1 25.1586,E2 457.0527} C_DIS
LIN {X 80.3612,Y -7.9572,Z 86,A -10.6088,B 24.9059,C -2.2396,E1 25.1591,E2 455.2524} C_DIS
LIN {X 80.576,Y -5.3442,Z 86,A -8.6922,B 24.9053,C -2.2474,E1 25.1595,E2 453.3288} C_DIS
LIN {X 80.6999,Y -2.9672,Z 86,A -7.0878,B 24.905,C -2.25,E1 25.1597,E2 451.7276} C_DIS
LIN {X 80.7477,Y -1.029,Z 86,A -5.4502,B 24.9039,C -2.2629,E1 25.1597,E2 450.0693} C_DIS
LIN {X 80.7303,Y 1.9749,Z 86,A -3.6026,B 24.9041,C -2.2605,E1 25.1597,E2 448.2385} C_DIS
LIN {X 80.6594,Y 3.9122,Z 86,A -1.9993,B 24.9031,C -2.2723,E1 25.1595,E2 446.6168} C_DIS
LIN {X 80.4594,Y 6.8949,Z 86,A -0.1282,B 24.9033,C -2.2709,E1 25.1591,E2 444.7602} C_DIS
LIN {X 80.2625,Y 8.9002,Z 86,A 1.2896,B 24.9029,C -2.275,E1 25.1587,E2 443.341} C_DIS
LIN {X 80.0206,Y 10.8619,Z 86,A 2.6819,B 24.9026,C -2.2791,E1 25.1582,E2 441.9473} C_DIS
LIN {X 79.7367,Y 12.7791,Z 86,A 4.0477,B 24.9022,C -2.2831,E1 25.1576,E2 440.5801} C_DIS
LIN {X 79.3241,Y 15.1245,Z 86,A 5.8943,B 24.9013,C -2.2934,E1 25.1567,E2 438.7199} C_DIS
LIN {X 78.7999,Y 17.6585,Z 86,A 7.55,B 24.9013,C -2.2932,E1 25.1557,E2 437.0743} C_DIS
LIN {X 78.3345,Y 19.6214,Z 86,A 8.9715,B 24.901,C -2.2972,E1 25.1548,E2 435.6514} C_DIS
LIN {X 77.8301,Y 21.535,Z 86,A 10.3661,B 24.9006,C -2.3012,E1 25.1537,E2 434.2556} C_DIS
LIN {X 77.3274,Y 23.2727,Z 86,A 11.8315,B 24.8998,C -2.3109,E1 25.1526,E2 432.7755} C_DIS
LIN {X 76.3699,Y 26.2469,Z 86,A 13.8494,B 24.8998,C -2.3111,E1 25.1508,E2 430.7687} C_DIS
LIN {X 75.7063,Y 28.1036,Z 86,A 15.2334,B 24.8995,C -2.3147,E1 25.1495,E2 429.3839} C_DIS
LIN {X 74.9835,Y 29.9794,Z 86,A 16.6507,B 24.8991,C -2.3185,E1 25.148,E2 427.9654} C_DIS
LIN {X 74.2289,Y 31.8016,Z 86,A 18.0412,B 24.8988,C -2.3222,E1 25.1465,E2 426.5738} C_DIS
LIN {X 73.4353,Y 33.5933,Z 86,A 19.4228,B 24.8985,C -2.3259,E1 25.1449,E2 425.191} C_DIS
LIN {X 72.574,Y 35.4161,Z 86,A 20.8446,B 24.8982,C -2.3296,E1 25.1432,E2 423.7681} C_DIS
LIN {X 71.685,Y 37.1826,Z 86,A 22.2393,B 24.8979,C -2.3332,E1 25.1414,E2 422.3724} C_DIS
LIN {X 70.5518,Y 39.2874,Z 86,A 24.0718,B 24.8971,C -2.3421,E1 25.139,E2 420.5282} C_DIS
LIN {X 68.9655,Y 42.0097,Z 86,A 26.2365,B 24.8967,C -2.3458,E1 25.1359,E2 418.3661} C_DIS
LIN {X 67.7055,Y 44.0139,Z 86,A 27.8179,B 24.8967,C -2.347,E1 25.1335,E2 416.7898} C_DIS
LIN {X 66.4725,Y 45.8534,Z 86,A 29.5703,B 24.8958,C -2.3567,E1 25.1307,E2 415.0231} C_DIS
LIN {X 64.8904,Y 48.0674,Z 86,A 31.3018,B 24.8959,C -2.3551,E1 25.1279,E2 413.3037} C_DIS
LIN {X 63.6844,Y 49.6543,Z 86,A 32.9166,B 24.8951,C -2.3648,E1 25.1251,E2 411.6735} C_DIS
LIN {X 61.9233,Y 51.8327,Z 86,A 34.9142,B 24.8946,C -2.3698,E1 25.1216,E2 409.6733} C_DIS
LIN {X 59.9009,Y 54.1579,Z 86,A 37.0193,B 24.8944,C -2.3722,E1 25.1177,E2 407.5721} C_DIS
LIN {X 57.8727,Y 56.32,Z 86,A 39.1812,B 24.8938,C -2.3786,E1 25.1135,E2 405.4045} C_DIS
LIN {X 56.041,Y 58.1416,Z 86,A 40.8871,B 24.8938,C -2.3784,E1 25.1101,E2 403.706} C_DIS
LIN {X 53.8805,Y 60.1492,Z 86,A 42.9786,B 24.8935,C -2.3826,E1 25.1058,E2 401.6131} C_DIS
LIN {X 51.6189,Y 62.101,Z 86,A 45.0834,B 24.8932,C -2.3862,E1 25.1013,E2 399.508} C_DIS
LIN {X 49.3242,Y 63.9388,Z 86,A 47.1528,B 24.8929,C -2.3894,E1 25.0967,E2 397.4386} C_DIS
LIN {X 47.4234,Y 65.3619,Z 86,A 48.7182,B 24.8929,C -2.3887,E1 25.0932,E2 395.8805} C_DIS
LIN {X 45.7399,Y 66.5514,Z 86,A 50.4354,B 24.892,C -2.3989,E1 25.0893,E2 394.145} C_DIS
LIN {X 43.2096,Y 68.2218,Z 86,A 52.3293,B 24.8924,C -2.3944,E1 25.0849,E2 392.268} C_DIS
LIN {X 41.5288,Y 69.2577,Z 86,A 53.9663,B 24.8916,C -2.4037,E1 25.0809,E2 390.6141} C_DIS
LIN {X 38.9629,Y 70.733,Z 86,A 55.8194,B 24.892,C -2.3991,E1 25.0764,E2 388.7774} C_DIS
LIN {X 37.2274,Y 71.6615,Z 86,A 57.4529,B 24.8912,C -2.4081,E1 25.0724,E2 387.127} C_DIS
LIN {X 34.5562,Y 72.9871,Z 86,A 59.3248,B 24.8916,C -2.4033,E1 25.0677,E2 385.2715} C_DIS
LIN {X 32.7235,Y 73.8272,Z 86,A 60.7475,B 24.8915,C -2.4047,E1 25.0641,E2 383.849} C_DIS
LIN {X 30.9408,Y 74.5916,Z 86,A 62.1217,B 24.8914,C -2.4061,E1 25.0605,E2 382.4748} C_DIS
LIN {X 29.1048,Y 75.327,Z 86,A 63.5231,B 24.8912,C -2.4074,E1 25.0569,E2 381.0734} C_DIS
LIN {X 27.3551,Y 75.9793,Z 86,A 64.8557,B 24.8912,C -2.4088,E1 25.0534,E2 379.7401} C_DIS
LIN {X 25.3388,Y 76.6761,Z 86,A 66.3551,B 24.891,C -2.4097,E1 25.0494,E2 378.2417} C_DIS
LIN {X 23.4945,Y 77.2609,Z 86,A 67.9647,B 24.8903,C -2.4177,E1 25.0451,E2 376.6157} C_DIS
LIN {X 20.6143,Y 78.0789,Z 86,A 69.8468,B 24.8908,C -2.4119,E1 25.0401,E2 374.7505} C_DIS
LIN {X 18.6948,Y 78.5605,Z 86,A 71.2502,B 24.8908,C -2.4127,E1 25.0363,E2 373.3473} C_DIS
LIN {X 16.7267,Y 79.0032,Z 86,A 72.6792,B 24.8907,C -2.4133,E1 25.0324,E2 371.9187} C_DIS
LIN {X 14.7857,Y 79.3893,Z 86,A 74.0816,B 24.8907,C -2.4139,E1 25.0285,E2 370.5166} C_DIS
LIN {X 12.8503,Y 79.7254,Z 86,A 75.4726,B 24.8907,C -2.4143,E1 25.0247,E2 369.1262} C_DIS
LIN {X 10.8707,Y 80.0194,Z 86,A 76.8936,B 24.8906,C -2.4147,E1 25.0208,E2 367.7054} C_DIS
LIN {X 8.896,Y 80.263,Z 86,A 78.302,B 24.8906,C -2.4148,E1 25.0169,E2 366.2978} C_DIS
LIN {X 6.9663,Y 80.4532,Z 86,A 79.677,B 24.8906,C -2.4149,E1 25.013,E2 364.9233} C_DIS
LIN {X 4.9561,Y 80.6022,Z 86,A 81.1106,B 24.8906,C -2.4151,E1 25.009,E2 363.49} C_DIS
LIN {X 2.9813,Y 80.6994,Z 86,A 82.5138,B 24.8906,C -2.415,E1 25.0051,E2 362.0874} C_DIS
LIN {X 1.0432,Y 80.7474,Z 86,A 83.8908,B 24.8906,C -2.4148,E1 25.0013,E2 360.7109} C_DIS
LIN {X -1.6068,Y 80.7371,Z 86,A 85.839,B 24.8904,C -2.4164,E1 24.9958,E2 358.759} C_DIS
LIN {X -3.9217,Y 80.659,Z 86,A 87.4164,B 24.8906,C -2.4139,E1 24.9915,E2 357.1871} C_DIS
LIN {X -5.8959,Y 80.5387,Z 86,A 88.8406,B 24.8906,C -2.4139,E1 24.9875,E2 355.7624} C_DIS
LIN {X -8.6187,Y 80.292,Z 86,A 90.7977,B 24.8906,C -2.4135,E1 24.982,E2 353.8053} C_DIS
LIN {X -10.8503,Y 80.0221,Z 86,A 92.3587,B 24.8909,C -2.4116,E1 24.9777,E2 352.2477} C_DIS
LIN {X -12.7892,Y 79.7351,Z 86,A 93.7518,B 24.8909,C -2.4107,E1 24.9739,E2 350.8554} C_DIS
LIN {X -14.7769,Y 79.391,Z 86,A 95.1856,B 24.891,C -2.4097,E1 24.9699,E2 349.4227} C_DIS
LIN {X -16.7177,Y 79.0051,Z 86,A 96.5924,B 24.8911,C -2.4086,E1 24.9661,E2 348.0167} C_DIS
LIN {X -18.6349,Y 78.5748,Z 86,A 98.2512,B 24.8906,C -2.4147,E1 24.9615,E2 346.3412} C_DIS
LIN {X -21.5277,Y 77.8321,Z 86,A 100.112,B 24.8914,C -2.4054,E1 24.9566,E2 344.4998} C_DIS
LIN {X -23.3784,Y 77.296,Z 86,A 101.4845,B 24.8915,C -2.4041,E1 24.9529,E2 343.1282} C_DIS
LIN {X -25.285,Y 76.6936,Z 86,A 102.9066,B 24.8917,C -2.4025,E1 24.9491,E2 341.7072} C_DIS
LIN {X -27.1331,Y 76.0593,Z 86,A 104.2975,B 24.8918,C -2.4009,E1 24.9455,E2 340.3174} C_DIS
LIN {X -29.014,Y 75.362,Z 86,A 105.9833,B 24.8913,C -2.4063,E1 24.941,E2 338.6153} C_DIS
LIN {X -31.8161,Y 74.2228,Z 86,A 107.8766,B 24.8922,C -2.3963,E1 24.9362,E2 336.7414} C_DIS
LIN {X -34.0786,Y 73.2099,Z 86,A 109.7493,B 24.8922,C -2.3968,E1 24.9314,E2 334.8629} C_DIS
LIN {X -36.2951,Y 72.1383,Z 86,A 111.3941,B 24.8927,C -2.3912,E1 24.9273,E2 333.2271} C_DIS
LIN {X -38.0488,Y 71.2289,Z 86,A 112.8004,B 24.8929,C -2.389,E1 24.9239,E2 331.8221} C_DIS
LIN {X -39.7541,Y 70.2911,Z 86,A 114.391,B 24.8926,C -2.3924,E1 24.9199,E2 330.219} C_DIS
LIN {X -42.2445,Y 68.8227,Z 86,A 116.2527,B 24.8934,C -2.3835,E1 24.9155,E2 328.3726} C_DIS
LIN {X -43.9188,Y 67.7666,Z 86,A 117.6527,B 24.8936,C -2.3808,E1 24.9122,E2 326.9747} C_DIS
LIN {X -45.5042,Y 66.7119,Z 86,A 119.033,B 24.8938,C -2.3789,E1 24.909,E2 325.5941} C_DIS
LIN {X -48.0617,Y 64.8946,Z 86,A 121.2522,B 24.8942,C -2.3742,E1 24.904,E2 323.3785} C_DIS
LIN {X -50.0668,Y 63.359,Z 86,A 123.1678,B 24.8942,C -2.3738,E1 24.8998,E2 321.4569} C_DIS
LIN {X -52.3726,Y 61.4666,Z 86,A 125.2875,B 24.8947,C -2.3692,E1 24.8953,E2 319.3399} C_DIS
LIN {X -54.5961,Y 59.5005,Z 86,A 127.4045,B 24.8951,C -2.3647,E1 24.8909,E2 317.2252} C_DIS
LIN {X -56.7457,Y 57.454,Z 86,A 129.5186,B 24.8955,C -2.36,E1 24.8866,E2 315.1136} C_DIS
LIN {X -58.8053,Y 55.3442,Z 86,A 131.6342,B 24.8959,C -2.3555,E1 24.8825,E2 312.9996} C_DIS
LIN {X -60.8102,Y 53.1334,Z 86,A 133.7591,B 24.8963,C -2.3504,E1 24.8786,E2 310.8773} C_DIS
LIN {X -62.7218,Y 50.8627,Z 86,A 135.8783,B 24.8968,C -2.3453,E1 24.8748,E2 308.7605} C_DIS
LIN {X -64.5334,Y 48.5436,Z 86,A 137.9922,B 24.8972,C -2.3404,E1 24.8712,E2 306.6481} C_DIS
LIN {X -66.0032,Y 46.5278,Z 86,A 139.644,B 24.8979,C -2.3325,E1 24.8686,E2 305.0071} C_DIS
LIN {X -67.1228,Y 44.8974,Z 86,A 141.0569,B 24.8982,C -2.3289,E1 24.8664,E2 303.5958} C_DIS
LIN {X -68.245,Y 43.1724,Z 86,A 142.4973,B 24.8986,C -2.3243,E1 24.8642,E2 302.159} C_DIS
LIN {X -69.2777,Y 41.4953,Z 86,A 143.9154,B 24.8989,C -2.3209,E1 24.8621,E2 300.7418} C_DIS
LIN {X -70.249,Y 39.8289,Z 86,A 145.5483,B 24.8987,C -2.3239,E1 24.8599,E2 299.0933} C_DIS
LIN {X -71.6572,Y 37.2354,Z 86,A 147.4147,B 24.8997,C -2.3119,E1 24.8574,E2 297.2457} C_DIS
LIN {X -72.5425,Y 35.4797,Z 86,A 148.8201,B 24.9001,C -2.3081,E1 24.8557,E2 295.8419} C_DIS
LIN {X -73.3996,Y 33.6712,Z 86,A 150.2431,B 24.9004,C -2.3039,E1 24.854,E2 294.421} C_DIS
LIN {X -74.2243,Y 31.8125,Z 86,A 151.6997,B 24.9008,C -2.2999,E1 24.8524,E2 292.9658} C_DIS
LIN {X -74.9668,Y 30.0206,Z 86,A 153.0878,B 24.9011,C -2.2961,E1 24.8509,E2 291.5792} C_DIS
LIN {X -75.6475,Y 28.2602,Z 86,A 154.4465,B 24.9014,C -2.2925,E1 24.8496,E2 290.2214} C_DIS
LIN {X -76.3456,Y 26.317,Z 86,A 155.9152,B 24.9018,C -2.2881,E1 24.8482,E2 288.7549} C_DIS
LIN {X -76.972,Y 24.4246,Z 86,A 157.3359,B 24.9021,C -2.2839,E1 24.847,E2 287.3361} C_DIS
LIN {X -77.563,Y 22.4779,Z 86,A 158.7867,B 24.9025,C -2.2796,E1 24.8459,E2 285.8872} C_DIS
LIN {X -78.0796,Y 20.6115,Z 86,A 160.1726,B 24.9028,C -2.2756,E1 24.8448,E2 284.5028} C_DIS
LIN {X -78.5602,Y 18.6959,Z 86,A 161.5845,B 24.9032,C -2.2715,E1 24.8439,E2 283.0925} C_DIS
LIN {X -79.0021,Y 16.7317,Z 86,A 163.0225,B 24.9036,C -2.2672,E1 24.8431,E2 281.6562} C_DIS
LIN {X -79.3875,Y 14.795,Z 86,A 164.433,B 24.9039,C -2.263,E1 24.8423,E2 280.2474} C_DIS
LIN {X -79.7254,Y 12.85,Z 86,A 165.844,B 24.9043,C -2.2588,E1 24.8417,E2 278.838} C_DIS
LIN {X -80.0155,Y 10.8986,Z 86,A 167.4386,B 24.9043,C -2.2594,E1 24.841,E2 277.2325} C_DIS
LIN {X -80.3505,Y 8.06,Z 86,A 169.4893,B 24.9047,C -2.2535,E1 24.8404,E2 275.1835} C_DIS
LIN {X -80.6028,Y 4.9472,Z 86,A 171.5251,B 24.9057,C -2.2418,E1 24.84,E2 273.1635} C_DIS
LIN {X -80.6998,Y 2.9719,Z 86,A 172.9415,B 24.9061,C -2.2377,E1 24.8399,E2 271.7484} C_DIS
LIN {X -80.7477,Y 1.0317,Z 86,A 174.6011,B 24.9058,C -2.2406,E1 24.8398,E2 270.0719} C_DIS
LIN {X -80.7353,Y -1.7052,Z 86,A 176.3288,B 24.9068,C -2.2289,E1 24.8398,E2 268.3617} C_DIS
LIN {X -80.6586,Y -3.9297,Z 86,A 177.878,B 24.9073,C -2.2231,E1 24.84,E2 266.8171} C_DIS
LIN {X -80.49,Y -6.5119,Z 86,A 179.8064,B 24.9076,C -2.2197,E1 24.8404,E2 264.8851} C_DIS
LIN {X -80.2717,Y -8.813,Z 86,A -178.6202,B 24.9082,C -2.2128,E1 24.8409,E2 263.3189} C_DIS
LIN {X -80.0175,Y -10.8847,Z 86,A -177.1448,B 24.9086,C -2.208,E1 24.8414,E2 261.8461} C_DIS
LIN {X -79.739,Y -12.764,Z 86,A -175.7755,B 24.9089,C -2.2043,E1 24.842,E2 260.4773} C_DIS
LIN {X -79.395,Y -14.7545,Z 86,A -174.3337,B 24.9092,C -2.2001,E1 24.8427,E2 259.0371} C_DIS
LIN {X -79.0143,Y -16.6725,Z 86,A -172.9378,B 24.9095,C -2.1961,E1 24.8435,E2 257.6425} C_DIS
LIN {X -78.5984,Y -18.5331,Z 86,A -171.5732,B 24.9099,C -2.1923,E1 24.8443,E2 256.2791} C_DIS
LIN {X -78.127,Y -20.4286,Z 86,A -169.9509,B 24.9097,C -2.1942,E1 24.8455,E2 254.6426} C_DIS
LIN {X -77.2904,Y -23.3974,Z 86,A -167.9746,B 24.9107,C -2.1821,E1 24.847,E2 252.6838} C_DIS
LIN {X -76.6843,Y -25.3139,Z 86,A -166.5401,B 24.911,C -2.1781,E1 24.8482,E2 251.2507} C_DIS
LIN {X -75.9206,Y -27.5161,Z 86,A -164.7152,B 24.911,C -2.1777,E1 24.8499,E2 249.4163} C_DIS
LIN {X -74.9805,Y -29.9868,Z 86,A -162.9881,B 24.9118,C -2.1684,E1 24.8517,E2 247.7017} C_DIS
LIN {X -74.2232,Y -31.8152,Z 86,A -161.574,B 24.9121,C -2.1647,E1 24.8532,E2 246.2887} C_DIS
LIN {X -73.437,Y -33.5895,Z 86,A -160.1887,B 24.9124,C -2.161,E1 24.8548,E2 244.9045} C_DIS
LIN {X -72.4746,Y -35.6168,Z 86,A -158.4046,B 24.9124,C -2.1617,E1 24.857,E2 243.1093} C_DIS
LIN {X -71.236,Y -38.0353,Z 86,A -156.6483,B 24.9132,C -2.1519,E1 24.8592,E2 241.367} C_DIS
LIN {X -70.3265,Y -39.6908,Z 86,A -155.2985,B 24.9134,C -2.1485,E1 24.8611,E2 240.018} C_DIS
LIN {X -68.9238,Y -42.0783,Z 86,A -153.111,B 24.9134,C -2.1493,E1 24.8642,E2 237.8174} C_DIS
LIN {X -67.1669,Y -44.8314,Z 86,A -150.9906,B 24.9143,C -2.1381,E1 24.8674,E2 235.713} C_DIS
LIN {X -66.0272,Y -46.494,Z 86,A -149.5533,B 24.9145,C -2.1348,E1 24.8697,E2 234.2766} C_DIS
LIN {X -64.6442,Y -48.3962,Z 86,A -147.716,B 24.9145,C -2.1352,E1 24.8728,E2 232.4294} C_DIS
LIN {X -62.751,Y -50.8268,Z 86,A -145.4901,B 24.9148,C -2.1311,E1 24.8767,E2 230.2028} C_DIS
LIN {X -61.1599,Y -52.7326,Z 86,A -143.6988,B 24.9151,C -2.1279,E1 24.8799,E2 228.411} C_DIS
LIN {X -59.2029,Y -54.9204,Z 86,A -141.5886,B 24.9154,C -2.1241,E1 24.8839,E2 226.3006} C_DIS
LIN {X -57.1178,Y -57.0861,Z 86,A -139.4503,B 24.9157,C -2.1197,E1 24.8881,E2 224.1636} C_DIS
LIN {X -54.9671,Y -59.16,Z 86,A -137.3245,B 24.9161,C -2.1156,E1 24.8924,E2 222.0389} C_DIS
LIN {X -52.8755,Y -61.0354,Z 86,A -135.2996,B 24.9163,C -2.1126,E1 24.8966,E2 220.0132} C_DIS
LIN {X -50.4774,Y -63.0341,Z 86,A -133.1024,B 24.9167,C -2.108,E1 24.9014,E2 217.8186} C_DIS
LIN {X -48.103,Y -64.8644,Z 86,A -130.9121,B 24.9168,C -2.106,E1 24.9063,E2 215.6251} C_DIS
LIN {X -45.7213,Y -66.5643,Z 86,A -129.096,B 24.9177,C -2.0954,E1 24.9104,E2 213.828} C_DIS
LIN {X -44.0467,Y -67.6843,Z 86,A -127.6625,B 24.9178,C -2.0933,E1 24.9137,E2 212.3949} C_DIS
LIN {X -42.4102,Y -68.7213,Z 86,A -126.2858,B 24.918,C -2.0913,E1 24.917,E2 211.0186} C_DIS
LIN {X -40.3927,Y -69.925,Z 86,A -124.436,B 24.9178,C -2.0941,E1 24.9215,E2 209.1566} C_DIS
LIN {X -38.0608,Y -71.2226,Z 86,A -122.716,B 24.9183,C -2.0867,E1 24.9257,E2 207.4494} C_DIS
LIN {X -36.339,Y -72.1161,Z 86,A -121.3309,B 24.9185,C -2.0852,E1 24.9291,E2 206.064} C_DIS
LIN {X -34.5617,Y -72.9845,Z 86,A -119.9226,B 24.9185,C -2.0837,E1 24.9326,E2 204.6557} C_DIS
LIN {X -32.8048,Y -73.7906,Z 86,A -118.5445,B 24.9187,C -2.0824,E1 24.9361,E2 203.2773} C_DIS
LIN {X -30.3249,Y -74.8429,Z 86,A -116.5731,B 24.9187,C -2.0822,E1 24.9412,E2 201.302} C_DIS
LIN {X -28.1439,Y -75.6915,Z 86,A -114.969,B 24.9189,C -2.079,E1 24.9454,E2 199.7021} C_DIS
LIN {X -26.322,Y -76.3439,Z 86,A -113.3897,B 24.9186,C -2.0837,E1 24.9496,E2 198.1085} C_DIS
LIN {X -23.4741,Y -77.2672,Z 86,A -111.463,B 24.9191,C -2.0765,E1 24.9547,E2 196.1955} C_DIS
LIN {X -21.5368,Y -77.8296,Z 86,A -110.0333,B 24.9192,C -2.0755,E1 24.9586,E2 194.7658} C_DIS
LIN {X -19.6603,Y -78.3245,Z 86,A -108.6534,B 24.9192,C -2.0748,E1 24.9623,E2 193.3855} C_DIS
LIN {X -17.6978,Y -78.7913,Z 86,A -106.9965,B 24.9188,C -2.0807,E1 24.9668,E2 191.7127} C_DIS
LIN {X -14.7822,Y -79.39,Z 86,A -104.8679,B 24.9188,C -2.0803,E1 24.9727,E2 189.5825} C_DIS
LIN {X -11.8433,Y -79.8813,Z 86,A -102.993,B 24.9194,C -2.0728,E1 24.9778,E2 187.7238} C_DIS
LIN {X -9.2612,Y -80.2203,Z 86,A -101.0841,B 24.9194,C -2.0743,E1 24.9831,E2 185.81} C_DIS
LIN {X -6.5894,Y -80.4838,Z 86,A -99.0689,B 24.9191,C -2.0774,E1 24.9887,E2 183.7863} C_DIS
LIN {X -4.0169,Y -80.6542,Z 86,A -97.4075,B 24.9194,C -2.0726,E1 24.9933,E2 182.1361} C_DIS
LIN {X -2.0429,Y -80.7283,Z 86,A -96.0113,B 24.9194,C -2.0726,E1 24.9972,E2 180.7396} C_DIS
LIN {X 0.5155,Y -80.7513,Z 86,A -94.5348,B 24.9202,C -2.063,E1 25.0013,E2 179.2859} C_DIS
Enddeposition()
LIN {X 0.5964,Y -89.2054,Z 87,A -94.3872,B 24.9305,C -1.9258,E1 25.0008,E2 179.4638} C_DIS
Startdeposition()
$VEL.CP = VEL_PRINT
LIN {X -1.7604,Y -89.1921,Z 87,A -96.1042,B 24.931,C -1.9188,E1 24.996,E2 181.1974} C_DIS
LIN {X -4.8057,Y -89.08,Z 87,A -98.0594,B 24.931,C -1.9188,E1 24.9905,E2 183.1533} C_DIS
LIN {X -7.6541,Y -88.8821,Z 87,A -99.823,B 24.9308,C -1.921,E1 24.9856,E2 184.9122} C_DIS
LIN {X -9.833,Y -88.6675,Z 87,A -101.4132,B 24.9312,C -1.9152,E1 24.9812,E2 186.5171} C_DIS
LIN {X -12.6653,Y -88.3059,Z 87,A -103.1877,B 24.9311,C -1.9175,E1 24.9763,E2 188.2875} C_DIS
LIN {X -15.907,Y -87.7798,Z 87,A -105.2468,B 24.9309,C -1.9198,E1 24.9706,E2 190.3432} C_DIS
LIN {X -18.8958,Y -87.1853,Z 87,A -107.2046,B 24.9309,C -1.9206,E1 24.9652,E2 192.3014} C_DIS
LIN {X -21.6765,Y -86.5376,Z 87,A -109.1961,B 24.9311,C -1.9165,E1 24.9598,E2 194.3053} C_DIS
LIN {X -24.4343,Y -85.798,Z 87,A -110.8785,B 24.9307,C -1.9225,E1 24.9553,E2 195.9761} C_DIS
LIN {X -27.3504,Y -84.9134,Z 87,A -112.8374,B 24.9307,C -1.9238,E1 24.9501,E2 197.9352} C_DIS
LIN {X -30.0543,Y -83.9962,Z 87,A -114.8174,B 24.9308,C -1.9208,E1 24.9448,E2 199.9263} C_DIS
LIN {X -33.1256,Y -82.833,Z 87,A -116.9018,B 24.9306,C -1.9235,E1 24.9394,E2 202.0086} C_DIS
LIN {X -35.7588,Y -81.7291,Z 87,A -118.628,B 24.9303,C -1.9288,E1 24.935,E2 203.7262} C_DIS
LIN {X -38.5293,Y -80.4601,Z 87,A -120.5886,B 24.9301,C -1.931,E1 24.93,E2 205.6867} C_DIS
LIN {X -41.0852,Y -79.1873,Z 87,A -122.5411,B 24.9301,C -1.9296,E1 24.9252,E2 207.6478} C_DIS
LIN {X -43.5974,Y -77.8306,Z 87,A -124.2012,B 24.9296,C -1.9374,E1 24.9211,E2 209.294} C_DIS
LIN {X -45.8637,Y -76.5189,Z 87,A -126.0673,B 24.9299,C -1.9341,E1 24.9166,E2 211.1736} C_DIS
LIN {X -48.288,Y -75.0107,Z 87,A -127.7954,B 24.9294,C -1.9402,E1 24.9126,E2 212.8928} C_DIS
LIN {X -50.4696,Y -73.5625,Z 87,A -129.4108,B 24.9291,C -1.9449,E1 24.9088,E2 214.5023} C_DIS
LIN {X -52.6058,Y -72.0483,Z 87,A -131.1695,B 24.9291,C -1.9454,E1 24.9048,E2 216.266} C_DIS
LIN {X -54.5457,Y -70.5911,Z 87,A -132.7289,B 24.9289,C -1.9481,E1 24.9014,E2 217.8246} C_DIS
LIN {X -56.5949,Y -68.9611,Z 87,A -134.5363,B 24.9289,C -1.9473,E1 24.8974,E2 219.6406} C_DIS
LIN {X -58.7717,Y -67.1135,Z 87,A -136.1933,B 24.9283,C -1.9562,E1 24.8939,E2 221.2829} C_DIS
LIN {X -60.7172,Y -65.3609,Z 87,A -137.8822,B 24.928,C -1.9593,E1 24.8905,E2 222.9712} C_DIS
LIN {X -62.6081,Y -63.5497,Z 87,A -139.6814,B 24.928,C -1.9593,E1 24.8868,E2 224.778} C_DIS
LIN {X -64.9048,Y -61.2022,Z 87,A -141.7622,B 24.9276,C -1.9646,E1 24.8828,E2 226.855} C_DIS
LIN {X -66.8313,Y -59.0948,Z 87,A -143.5343,B 24.9272,C -1.9705,E1 24.8795,E2 228.6209} C_DIS
LIN {X -68.2614,Y -57.4369,Z 87,A -145.1324,B 24.9274,C -1.968,E1 24.8766,E2 230.2322} C_DIS
LIN {X -70.0633,Y -55.222,Z 87,A -146.8634,B 24.9268,C -1.9754,E1 24.8736,E2 231.9537} C_DIS
LIN {X -71.655,Y -53.143,Z 87,A -148.6666,B 24.9268,C -1.9759,E1 24.8706,E2 233.7645} C_DIS
LIN {X -73.3177,Y -50.8218,Z 87,A -150.398,B 24.9262,C -1.9835,E1 24.8678,E2 235.4863} C_DIS
LIN {X -75.0107,Y -48.288,Z 87,A -152.365,B 24.9259,C -1.9882,E1 24.8648,E2 237.452} C_DIS
LIN {X -76.5189,Y -45.8637,Z 87,A -154.1383,B 24.9254,C -1.9947,E1 24.8622,E2 239.2187} C_DIS
LIN {X -77.8306,Y -43.5974,Z 87,A -155.9011,B 24.9252,C -1.9969,E1 24.8598,E2 240.9856} C_DIS
LIN {X -79.1873,Y -41.0852,Z 87,A -157.8601,B 24.9252,C -1.9982,E1 24.8572,E2 242.952} C_DIS
LIN {X -80.4601,Y -38.5293,Z 87,A -159.5927,B 24.9245,C -2.0062,E1 24.8551,E2 244.6746} C_DIS
LIN {X -81.5577,Y -36.152,Z 87,A -161.3889,B 24.9245,C -2.0076,E1 24.853,E2 246.4774} C_DIS
LIN {X -82.6713,Y -33.5229,Z 87,A -163.1305,B 24.9238,C -2.0156,E1 24.8511,E2 248.2097} C_DIS
LIN {X -83.621,Y -31.0828,Z 87,A -164.7506,B 24.9233,C -2.0222,E1 24.8495,E2 249.823} C_DIS
LIN {X -84.3587,Y -29.0213,Z 87,A -166.3785,B 24.9235,C -2.0199,E1 24.848,E2 251.4656} C_DIS
LIN {X -85.3697,Y -25.8966,Z 87,A -168.2892,B 24.9226,C -2.032,E1 24.8464,E2 253.3586} C_DIS
LIN {X -85.9795,Y -23.7937,Z 87,A -169.7051,B 24.9223,C -2.0359,E1 24.8454,E2 254.7733} C_DIS
LIN {X -86.5376,Y -21.6765,Z 87,A -171.1209,B 24.922,C -2.0399,E1 24.8444,E2 256.1877} C_DIS
LIN {X -87.181,Y -18.9159,Z 87,A -172.9588,B 24.9216,C -2.0451,E1 24.8432,E2 258.0242} C_DIS
LIN {X -87.7039,Y -16.3292,Z 87,A -174.6604,B 24.9212,C -2.0501,E1 24.8423,E2 259.7239} C_DIS
LIN {X -88.0782,Y -14.1719,Z 87,A -176.2617,B 24.9212,C -2.0488,E1 24.8416,E2 261.3378} C_DIS
LIN {X -88.4851,Y -11.3458,Z 87,A -177.923,B 24.9205,C -2.0596,E1 24.841,E2 262.9833} C_DIS
LIN {X -88.7369,Y -9.1709,Z 87,A -179.4116,B 24.9203,C -2.0616,E1 24.8405,E2 264.4759} C_DIS
LIN {X -88.9983,Y -6.1348,Z 87,A 178.6185,B 24.9198,C -2.0675,E1 24.8401,E2 266.4437} C_DIS
LIN {X -89.1506,Y -3.2836,Z 87,A 176.6579,B 24.9197,C -2.0696,E1 24.8398,E2 268.411} C_DIS
LIN {X -89.2126,Y -0.0065,Z 87,A 174.4253,B 24.9194,C -2.0727,E1 24.8398,E2 270.6498} C_DIS
LIN {X -89.1506,Y 3.2836,Z 87,A 172.5945,B 24.9183,C -2.0876,E1 24.8399,E2 272.456} C_DIS
LIN {X -89.0432,Y 5.4705,Z 87,A 170.9929,B 24.9183,C -2.0865,E1 24.8402,E2 274.0699} C_DIS
LIN {X -88.821,Y 8.3171,Z 87,A 169.2584,B 24.9177,C -2.0952,E1 24.8406,E2 275.794} C_DIS
LIN {X -88.5402,Y 10.9204,Z 87,A 167.6378,B 24.9171,C -2.1023,E1 24.8411,E2 277.4073} C_DIS
LIN {X -88.18,Y 13.5139,Z 87,A 165.8726,B 24.9169,C -2.1053,E1 24.8418,E2 279.1759} C_DIS
LIN {X -87.7798,Y 15.907,Z 87,A 164.3745,B 24.9163,C -2.112,E1 24.8425,E2 280.6669} C_DIS
LIN {X -87.2768,Y 18.4766,Z 87,A 162.4956,B 24.9163,C -2.1116,E1 24.8436,E2 282.5577} C_DIS
LIN {X -86.6392,Y 21.2598,Z 87,A 160.7615,B 24.9157,C -2.1203,E1 24.8447,E2 284.2813} C_DIS
LIN {X -85.8062,Y 24.4053,Z 87,A 158.6479,B 24.9152,C -2.1262,E1 24.8462,E2 286.3931} C_DIS
LIN {X -84.9134,Y 27.3504,Z 87,A 156.6681,B 24.9147,C -2.1322,E1 24.8479,E2 288.3699} C_DIS
LIN {X -83.9962,Y 30.0543,Z 87,A 154.893,B 24.9141,C -2.1395,E1 24.8495,E2 290.1376} C_DIS
LIN {X -83.0999,Y 32.4464,Z 87,A 153.1466,B 24.914,C -2.1415,E1 24.8513,E2 291.8891} C_DIS
LIN {X -81.9952,Y 35.1485,Z 87,A 151.3535,B 24.9133,C -2.1495,E1 24.8532,E2 293.673} C_DIS
LIN {X -81.1079,Y 37.1501,Z 87,A 149.7526,B 24.9135,C -2.1481,E1 24.855,E2 295.2861} C_DIS
LIN {X -79.876,Y 39.726,Z 87,A 148.0919,B 24.9126,C -2.1586,E1 24.857,E2 296.9308} C_DIS
LIN {X -78.6772,Y 42.0538,Z 87,A 146.3994,B 24.9122,C -2.1632,E1 24.8592,E2 298.6214} C_DIS
LIN {X -77.6214,Y 43.972,Z 87,A 144.7989,B 24.9124,C -2.1616,E1 24.8614,E2 300.2341} C_DIS
LIN {X -76.1731,Y 46.4326,Z 87,A 143.066,B 24.9117,C -2.1697,E1 24.8639,E2 301.9564} C_DIS
LIN {X -74.7949,Y 48.6241,Z 87,A 141.2786,B 24.9117,C -2.1708,E1 24.8666,E2 303.7505} C_DIS
LIN {X -73.1212,Y 51.1045,Z 87,A 139.3003,B 24.9113,C -2.1744,E1 24.8697,E2 305.7298} C_DIS
LIN {X -71.2551,Y 53.6753,Z 87,A 137.4067,B 24.9105,C -2.1842,E1 24.8729,E2 307.6093} C_DIS
LIN {X -69.6504,Y 55.7444,Z 87,A 135.6028,B 24.9105,C -2.185,E1 24.876,E2 309.4197} C_DIS
LIN {X -67.8296,Y 57.9437,Z 87,A 133.9432,B 24.9096,C -2.1948,E1 24.8789,E2 311.0635} C_DIS
LIN {X -66.1011,Y 59.9105,Z 87,A 132.0671,B 24.9098,C -2.1933,E1 24.8825,E2 312.9515} C_DIS
LIN {X -64.1488,Y 61.994,Z 87,A 130.3359,B 24.9091,C -2.2009,E1 24.8858,E2 314.6723} C_DIS
LIN {X -62.3029,Y 63.8511,Z 87,A 128.5328,B 24.9091,C -2.2013,E1 24.8894,E2 316.482} C_DIS
LIN {X -60.2266,Y 65.811,Z 87,A 126.8746,B 24.9083,C -2.2107,E1 24.8927,E2 318.1244} C_DIS
LIN {X -58.2703,Y 67.5514,Z 87,A 124.9994,B 24.9085,C -2.2088,E1 24.8967,E2 320.0117} C_DIS
LIN {X -56.0777,Y 69.3803,Z 87,A 123.2691,B 24.9079,C -2.2159,E1 24.9004,E2 321.7316} C_DIS
LIN {X -53.6753,Y 71.2551,Z 87,A 121.3039,B 24.9076,C -2.2197,E1 24.9047,E2 323.6948} C_DIS
LIN {X -51.6407,Y 72.7434,Z 87,A 119.5147,B 24.9077,C -2.218,E1 24.9088,E2 325.4944} C_DIS
LIN {X -49.0072,Y 74.5428,Z 87,A 117.6188,B 24.907,C -2.2265,E1 24.9132,E2 327.3763} C_DIS
LIN {X -46.7992,Y 75.9503,Z 87,A 116.0024,B 24.9066,C -2.2316,E1 24.917,E2 328.9858} C_DIS
LIN {X -44.9212,Y 77.076,Z 87,A 114.4058,B 24.9069,C -2.2284,E1 24.9209,E2 330.5948} C_DIS
LIN {X -42.4309,Y 78.4726,Z 87,A 112.6774,B 24.9063,C -2.2347,E1 24.9251,E2 332.3131} C_DIS
LIN {X -39.726,Y 79.876,Z 87,A 110.7145,B 24.9061,C -2.2377,E1 24.9299,E2 334.2741} C_DIS
LIN {X -37.1501,Y 81.1079,Z 87,A 108.7609,B 24.9061,C -2.2368,E1 24.9349,E2 336.2346} C_DIS
LIN {X -34.5349,Y 82.2537,Z 87,A 107.1056,B 24.9055,C -2.2449,E1 24.9391,E2 337.8746} C_DIS
LIN {X -32.1066,Y 83.2333,Z 87,A 105.2341,B 24.9058,C -2.2414,E1 24.944,E2 339.7585} C_DIS
LIN {X -29.4261,Y 84.2166,Z 87,A 103.5076,B 24.9053,C -2.247,E1 24.9485,E2 341.4751} C_DIS
LIN {X -26.9423,Y 85.0455,Z 87,A 101.6857,B 24.9055,C -2.2447,E1 24.9534,E2 343.3059} C_DIS
LIN {X -23.7937,Y 85.9795,Z 87,A 99.7793,B 24.9048,C -2.2532,E1 24.9584,E2 345.1952} C_DIS
LIN {X -21.6765,Y 86.5376,Z 87,A 98.1856,B 24.9051,C -2.2488,E1 24.9628,E2 346.8017} C_DIS
LIN {X -18.9055,Y 87.1832,Z 87,A 96.5367,B 24.9045,C -2.2559,E1 24.9672,E2 348.4356} C_DIS
LIN {X -16.3292,Y 87.7039,Z 87,A 94.8478,B 24.9045,C -2.2572,E1 24.9719,E2 350.1233} C_DIS
LIN {X -14.1719,Y 88.0782,Z 87,A 93.4394,B 24.9043,C -2.2582,E1 24.9757,E2 351.5308} C_DIS
LIN {X -11.5807,Y 88.4546,Z 87,A 91.6844,B 24.9044,C -2.257,E1 24.9806,E2 353.29} C_DIS
LIN {X -9.1709,Y 88.7369,Z 87,A 90.1951,B 24.9042,C -2.26,E1 24.9847,E2 354.7731} C_DIS
LIN {X -6.9904,Y 88.9352,Z 87,A 88.715,B 24.9043,C -2.2583,E1 24.9889,E2 356.2578} C_DIS
LIN {X -3.8277,Y 89.1273,Z 87,A 86.7196,B 24.9042,C -2.2603,E1 24.9944,E2 358.249} C_DIS
LIN {X -1.0948,Y 89.2044,Z 87,A 84.8123,B 24.9045,C -2.256,E1 24.9998,E2 360.1668} C_DIS
LIN {X 1.7604,Y 89.1921,Z 87,A 83.0867,B 24.9042,C -2.2597,E1 25.0046,E2 361.8834} C_DIS
LIN {X 4.3774,Y 89.1036,Z 87,A 81.2504,B 24.9046,C -2.2548,E1 25.0097,E2 363.7307} C_DIS
LIN {X 7.6541,Y 88.8821,Z 87,A 79.1837,B 24.9046,C -2.2561,E1 25.0155,E2 365.7933} C_DIS
LIN {X 10.761,Y 88.5589,Z 87,A 77.3498,B 24.9041,C -2.2613,E1 25.0205,E2 367.6136} C_DIS
LIN {X 13.5139,Y 88.18,Z 87,A 75.5079,B 24.9043,C -2.259,E1 25.0256,E2 369.4593} C_DIS
LIN {X 15.907,Y 87.7798,Z 87,A 74.0212,B 24.9041,C -2.2608,E1 25.0297,E2 370.9402} C_DIS
LIN {X 18.4766,Y 87.2768,Z 87,A 72.1191,B 24.9048,C -2.2529,E1 25.0349,E2 372.8588} C_DIS
LIN {X 21.2598,Y 86.6392,Z 87,A 70.4374,B 24.9045,C -2.2568,E1 25.0395,E2 374.5287} C_DIS
LIN {X 24.2065,Y 85.8626,Z 87,A 68.4843,B 24.9045,C -2.2557,E1 25.0447,E2 376.4814} C_DIS
LIN {X 26.5325,Y 85.1725,Z 87,A 66.9271,B 24.9046,C -2.2546,E1 25.0489,E2 378.0384} C_DIS
LIN {X 29.0213,Y 84.3587,Z 87,A 65.0784,B 24.9052,C -2.2477,E1 25.0538,E2 379.8999} C_DIS
LIN {X 32.1066,Y 83.2333,Z 87,A 63.2156,B 24.9047,C -2.2538,E1 25.0586,E2 381.7442} C_DIS
LIN {X 34.5349,Y 82.2537,Z 87,A 61.4669,B 24.905,C -2.2499,E1 25.0632,E2 383.4981} C_DIS
LIN {X 37.1501,Y 81.1079,Z 87,A 59.7081,B 24.905,C -2.2503,E1 25.0676,E2 385.2517} C_DIS
LIN {X 39.1294,Y 80.1717,Z 87,A 58.3059,B 24.9051,C -2.2487,E1 25.0712,E2 386.6539} C_DIS
LIN {X 41.4647,Y 78.9874,Z 87,A 56.558,B 24.9055,C -2.2444,E1 25.0755,E2 388.4073} C_DIS
LIN {X 43.5974,Y 77.8306,Z 87,A 55.0032,B 24.9057,C -2.2423,E1 25.0793,E2 389.9624} C_DIS
LIN {X 46.2303,Y 76.2961,Z 87,A 53.0535,B 24.9059,C -2.2397,E1 25.084,E2 391.9122} C_DIS
LIN {X 48.649,Y 74.7789,Z 87,A 51.2964,B 24.9059,C -2.2394,E1 25.0881,E2 393.6644} C_DIS
LIN {X 50.4696,Y 73.5625,Z 87,A 49.7118,B 24.9066,C -2.2311,E1 25.0918,E2 395.2632} C_DIS
LIN {X 52.9683,Y 71.7829,Z 87,A 47.9109,B 24.9064,C -2.2335,E1 25.0959,E2 397.0522} C_DIS
LIN {X 54.8585,Y 70.3501,Z 87,A 46.2295,B 24.9071,C -2.2254,E1 25.0996,E2 398.7466} C_DIS
LIN {X 57.107,Y 68.5356,Z 87,A 44.4948,B 24.9071,C -2.2261,E1 25.1034,E2 400.4731} C_DIS
LIN {X 59.0948,Y 66.8313,Z 87,A 42.892,B 24.9071,C -2.2254,E1 25.1067,E2 402.071} C_DIS
LIN {X 60.7172,Y 65.3609,Z 87,A 41.3092,B 24.9078,C -2.2166,E1 25.11,E2 403.6684} C_DIS
LIN {X 62.7766,Y 63.3832,Z 87,A 39.5948,B 24.9078,C -2.2169,E1 25.1134,E2 405.375} C_DIS
LIN {X 64.9581,Y 61.1454,Z 87,A 37.5468,B 24.9083,C -2.2111,E1 25.1174,E2 407.4278} C_DIS
LIN {X 66.8313,Y 59.0948,Z 87,A 35.8938,B 24.9083,C -2.2116,E1 25.1205,E2 409.0722} C_DIS
LIN {X 68.2614,Y 57.4369,Z 87,A 34.4946,B 24.9085,C -2.2086,E1 25.123,E2 410.4722} C_DIS
LIN {X 69.9164,Y 55.4078,Z 87,A 32.7514,B 24.909,C -2.2025,E1 25.1261,E2 412.2217} C_DIS
LIN {X 71.655,Y 53.143,Z 87,A 30.8016,B 24.9097,C -2.194,E1 25.1294,E2 414.1822} C_DIS
LIN {X 73.5625,Y 50.4696,Z 87,A 28.8997,B 24.9095,C -2.1959,E1 25.1324,E2 416.0703} C_DIS
LIN {X 75.0107,Y 48.288,Z 87,A 27.157,B 24.9101,C -2.1895,E1 25.1351,E2 417.8194} C_DIS
LIN {X 76.5189,Y 45.8637,Z 87,A 25.295,B 24.9106,C -2.1837,E1 25.1378,E2 419.6857} C_DIS
LIN {X 77.946,Y 43.3907,Z 87,A 23.5808,B 24.9106,C -2.183,E1 25.1401,E2 421.3927} C_DIS
LIN {X 78.9874,Y 41.4647,Z 87,A 22.183,B 24.9109,C -2.1795,E1 25.142,E2 422.7914} C_DIS
LIN {X 80.1717,Y 39.1294,Z 87,A 20.3289,B 24.9118,C -2.1687,E1 25.1443,E2 424.661} C_DIS
LIN {X 81.3814,Y 36.5431,Z 87,A 18.6892,B 24.9116,C -2.1704,E1 25.1462,E2 426.2879} C_DIS
LIN {X 82.2537,Y 34.5349,Z 87,A 17.2199,B 24.9122,C -2.1642,E1 25.1478,E2 427.7639} C_DIS
LIN {X 83.2813,Y 31.98,Z 87,A 15.3454,B 24.9129,C -2.1553,E1 25.1497,E2 429.649} C_DIS
LIN {X 84.3587,Y 29.0213,Z 87,A 13.5248,B 24.9128,C -2.1564,E1 25.1514,E2 431.4566} C_DIS
LIN {X 85.1725,Y 26.5325,Z 87,A 11.7838,B 24.9134,C -2.1493,E1 25.1529,E2 433.2045} C_DIS
LIN {X 85.9795,Y 23.7937,Z 87,A 10.0321,B 24.9136,C -2.1467,E1 25.1543,E2 434.9525} C_DIS
LIN {X 86.5376,Y 21.6765,Z 87,A 8.432,B 24.9145,C -2.1355,E1 25.1554,E2 436.5696} C_DIS
LIN {X 87.2768,Y 18.4766,Z 87,A 6.5403,B 24.9144,C -2.1367,E1 25.1565,E2 438.4475} C_DIS
LIN {X 87.8014,Y 15.7873,Z 87,A 4.6851,B 24.9151,C -2.1279,E1 25.1575,E2 440.3126} C_DIS
LIN {X 88.2455,Y 13.09,Z 87,A 2.8659,B 24.9157,C -2.1201,E1 25.1583,E2 442.1394} C_DIS
LIN {X 88.6176,Y 10.2591,Z 87,A 1.2274,B 24.9157,C -2.1213,E1 25.1588,E2 443.7655} C_DIS
LIN {X 88.871,Y 7.7742,Z 87,A -0.5588,B 24.9165,C -2.1098,E1 25.1593,E2 445.5685} C_DIS
LIN {X 89.08,Y 4.8057,Z 87,A -2.3354,B 24.9166,C -2.1085,E1 25.1596,E2 447.3375} C_DIS
LIN {X 89.1921,Y 1.7604,Z 87,A -4.3078,B 24.9172,C -2.1017,E1 25.1598,E2 449.3142} C_DIS
LIN {X 89.1921,Y -1.7604,Z 87,A -6.5247,B 24.9176,C -2.096,E1 25.1598,E2 451.5313} C_DIS
LIN {X 89.08,Y -4.8057,Z 87,A -8.4666,B 24.9181,C -2.0903,E1 25.1595,E2 453.4752} C_DIS
LIN {X 88.8821,Y -7.6541,Z 87,A -10.2177,B 24.9183,C -2.0873,E1 25.1591,E2 455.2229} C_DIS
LIN {X 88.6675,Y -9.833,Z 87,A -11.6139,B 24.9186,C -2.0832,E1 25.1587,E2 456.6206} C_DIS
LIN {X 88.3995,Y -12.0061,Z 87,A -13.1928,B 24.9194,C -2.0725,E1 25.1581,E2 458.2153} C_DIS
LIN {X 87.9684,Y -14.8286,Z 87,A -14.8315,B 24.9194,C -2.0736,E1 25.1574,E2 459.8418} C_DIS
LIN {X 87.578,Y -16.983,Z 87,A -16.2993,B 24.9199,C -2.067,E1 25.1567,E2 461.3167} C_DIS
LIN {X 87.0435,Y -19.5463,Z 87,A -18.0725,B 24.9206,C -2.0583,E1 25.1556,E2 463.1} C_DIS
LIN {X 86.3718,Y -22.3214,Z 87,A -19.7167,B 24.9205,C -2.0593,E1 25.1545,E2 464.7324} C_DIS
LIN {X 85.798,Y -24.4343,Z 87,A -21.1159,B 24.9208,C -2.0551,E1 25.1534,E2 466.1334} C_DIS
LIN {X 85.1725,Y -26.5325,Z 87,A -22.5839,B 24.9213,C -2.0486,E1 25.1522,E2 467.6085} C_DIS
LIN {X 84.2166,Y -29.4261,Z 87,A -24.5266,B 24.9217,C -2.043,E1 25.1505,E2 469.5534} C_DIS
LIN {X 83.3852,Y -31.7055,Z 87,A -26.004,B 24.9219,C -2.0411,E1 25.1491,E2 471.0271} C_DIS
LIN {X 82.4203,Y -34.1396,Z 87,A -27.6745,B 24.9222,C -2.0363,E1 25.1473,E2 472.6996} C_DIS
LIN {X 81.5577,Y -36.152,Z 87,A -29.2631,B 24.9231,C -2.0256,E1 25.1455,E2 474.3048} C_DIS
LIN {X 80.1717,Y -39.1294,Z 87,A -31.3494,B 24.9235,C -2.0201,E1 25.143,E2 476.3929} C_DIS
LIN {X 78.8771,Y -41.6743,Z 87,A -33.0609,B 24.9235,C -2.0191,E1 25.1408,E2 478.0978} C_DIS
LIN {X 77.5896,Y -44.0273,Z 87,A -34.9178,B 24.9243,C -2.0093,E1 25.1383,E2 479.968} C_DIS
LIN {X 75.897,Y -46.8846,Z 87,A -37.0211,B 24.9247,C -2.0042,E1 25.1352,E2 482.0726} C_DIS
LIN {X 74.1763,Y -49.563,Z 87,A -38.8994,B 24.9247,C -2.0044,E1 25.1324,E2 483.9412} C_DIS
LIN {X 72.5509,Y -51.9105,Z 87,A -40.7472,B 24.9251,C -1.9989,E1 25.1294,E2 485.7929} C_DIS
LIN {X 71.0123,Y -53.9986,Z 87,A -42.5158,B 24.9257,C -1.9907,E1 25.1264,E2 487.5723} C_DIS
LIN {X 69.2312,Y -56.2617,Z 87,A -44.1707,B 24.9255,C -1.9927,E1 25.1236,E2 489.2148} C_DIS
LIN {X 67.5514,Y -58.2703,Z 87,A -45.8426,B 24.9258,C -1.9887,E1 25.1205,E2 490.8886} C_DIS
LIN {X 65.811,Y -60.2266,Z 87,A -47.5855,B 24.9263,C -1.9823,E1 25.1173,E2 492.6389} C_DIS
LIN {X 64.1488,Y -61.994,Z 87,A -49.1368,B 24.9266,C -1.9787,E1 25.1143,E2 494.1919} C_DIS
LIN {X 62.3029,Y -63.8511,Z 87,A -50.9208,B 24.9272,C -1.971,E1 25.1107,E2 495.9865} C_DIS
LIN {X 60.2266,Y -65.811,Z 87,A -52.6855,B 24.9272,C -1.9692,E1 25.1071,E2 497.7484} C_DIS
LIN {X 57.7635,Y -67.9832,Z 87,A -54.8616,B 24.9278,C -1.9621,E1 25.1025,E2 499.9328} C_DIS
LIN {X 55.222,Y -70.0633,Z 87,A -56.8321,B 24.9278,C -1.9623,E1 25.0982,E2 501.8954} C_DIS
LIN {X 53.143,Y -71.655,Z 87,A -58.6173,B 24.9283,C -1.9551,E1 25.0942,E2 503.691} C_DIS
LIN {X 50.8218,Y -73.3177,Z 87,A -60.3317,B 24.9283,C -1.9555,E1 25.0903,E2 505.3985} C_DIS
LIN {X 48.288,Y -75.0107,Z 87,A -62.2793,B 24.9286,C -1.952,E1 25.0858,E2 507.3479} C_DIS
LIN {X 45.8637,Y -76.5189,Z 87,A -64.0352,B 24.9286,C -1.9513,E1 25.0816,E2 509.1001} C_DIS
LIN {X 43.5974,Y -77.8306,Z 87,A -65.7806,B 24.929,C -1.9461,E1 25.0773,E2 510.8526} C_DIS
LIN {X 41.0852,Y -79.1873,Z 87,A -67.7205,B 24.9295,C -1.9393,E1 25.0725,E2 512.803} C_DIS
LIN {X 38.5293,Y -80.4601,Z 87,A -69.4365,B 24.9295,C -1.9404,E1 25.0682,E2 514.5119} C_DIS
LIN {X 35.7588,Y -81.7291,Z 87,A -71.3859,B 24.9296,C -1.9377,E1 25.0633,E2 516.4628} C_DIS
LIN {X 33.1256,Y -82.833,Z 87,A -73.3319,B 24.9301,C -1.9313,E1 25.0582,E2 518.4197} C_DIS
LIN {X 30.0543,Y -83.9962,Z 87,A -75.43,B 24.9303,C -1.9288,E1 25.0527,E2 520.519} C_DIS
LIN {X 27.3504,Y -84.9134,Z 87,A -77.1475,B 24.9301,C -1.9305,E1 25.0482,E2 522.2292} C_DIS
LIN {X 24.4343,Y -85.798,Z 87,A -79.171,B 24.9304,C -1.9261,E1 25.0427,E2 524.2598} C_DIS
LIN {X 21.6765,Y -86.5376,Z 87,A -81.0412,B 24.9307,C -1.923,E1 25.0377,E2 526.1345} C_DIS
LIN {X 18.8958,Y -87.1853,Z 87,A -82.6877,B 24.9303,C -1.9276,E1 25.0332,E2 527.7679} C_DIS
LIN {X 16.3292,Y -87.7039,Z 87,A -84.55,B 24.9309,C -1.9201,E1 25.0281,E2 529.6456} C_DIS
LIN {X 13.5139,Y -88.18,Z 87,A -86.2693,B 24.9307,C -1.9226,E1 25.0234,E2 531.3574} C_DIS
LIN {X 10.9204,Y -88.5402,Z 87,A -88.0883,B 24.9311,C -1.9169,E1 25.0183,E2 533.1883} C_DIS
LIN {X 7.6541,Y -88.8821,Z 87,A -90.1672,B 24.9311,C -1.9169,E1 25.0125,E2 535.2662} C_DIS
LIN {X 4.8057,Y -89.08,Z 87,A -91.8155,B 24.9307,C -1.9222,E1 25.008,E2 536.9012} C_DIS
LIN {X 2.6181,Y -89.1711,Z 87,A -93.2887,B 24.9309,C -1.9195,E1 25.0038,E2 538.3804} C_DIS
LIN {X 0.5964,Y -89.2054,Z 87,A -94.387,B 24.9305,C -1.9257,E1 25.0008,E2 539.4638} C_DIS
Enddeposition()
LIN {X 0.5964,Y -89.2054,Z 87,A -94.387,B 24.9305,C -1.9257,E1 25.0008,E2 539.4638} C_DIS
Startdeposition()
$VEL.CP = VEL_PRINT
LIN {X 1.3805,Y -88.305,Z 87,A -93.3645,B 24.9281,C -1.9582,E1 25.0039,E2 538.3643} C_DIS
LIN {X 4.5019,Y -88.2014,Z 87,A -91.1847,B 24.9277,C -1.964,E1 25.01,E2 536.1714} C_DIS
LIN {X 7.9332,Y -87.9586,Z 87,A -88.9964,B 24.9277,C -1.9637,E1 25.0161,E2 533.985} C_DIS
LIN {X 11.3287,Y -87.5858,Z 87,A -86.4903,B 24.9269,C -1.9747,E1 25.0231,E2 531.4548} C_DIS
LIN {X 15.9861,Y -86.8573,Z 87,A -83.232,B 24.9262,C -1.9837,E1 25.0321,E2 528.1784} C_DIS
LIN {X 20.5572,Y -85.8904,Z 87,A -80.6902,B 24.9272,C -1.9701,E1 25.0389,E2 525.6725} C_DIS
LIN {X 23.6094,Y -85.1026,Z 87,A -78.6645,B 24.9272,C -1.9716,E1 25.0444,E2 523.6464} C_DIS
LIN {X 27.1221,Y -84.0477,Z 87,A -76.2519,B 24.9268,C -1.9755,E1 25.0508,E2 521.2289} C_DIS
LIN {X 30.606,Y -82.8434,Z 87,A -74.0583,B 24.9271,C -1.9718,E1 25.0566,E2 519.0484} C_DIS
LIN {X 32.3809,Y -82.1651,Z 87,A -72.0739,B 24.9251,C -1.9992,E1 25.0619,E2 517.0036} C_DIS
LIN {X 35.7075,Y -80.7762,Z 87,A -70.2892,B 24.9262,C -1.9837,E1 25.0664,E2 515.26} C_DIS
LIN {X 38.6741,Y -79.3987,Z 87,A -68.1632,B 24.926,C -1.9872,E1 25.0717,E2 513.1312} C_DIS
LIN {X 41.6745,Y -77.8659,Z 87,A -65.642,B 24.9248,C -2.0024,E1 25.078,E2 510.5811} C_DIS
LIN {X 45.4586,Y -75.719,Z 87,A -63.1451,B 24.9253,C -1.9963,E1 25.084,E2 508.1063} C_DIS
LIN {X 48.4083,Y -73.8669,Z 87,A -60.9532,B 24.9251,C -1.9983,E1 25.0891,E2 505.9167} C_DIS
LIN {X 53.2151,Y -70.4827,Z 87,A -57.1043,B 24.9244,C -2.0073,E1 25.0979,E2 502.0601} C_DIS
LIN {X 56.3649,Y -67.9898,Z 87,A -54.5409,B 24.9241,C -2.0115,E1 25.1034,E2 499.4964} C_DIS
LIN {X 58.457,Y -66.2014,Z 87,A -52.4969,B 24.9231,C -2.0247,E1 25.1078,E2 497.4295} C_DIS
LIN {X 61.6067,Y -63.2806,Z 87,A -49.9867,B 24.9234,C -2.0215,E1 25.1128,E2 494.937} C_DIS
LIN {X 63.3132,Y -61.5728,Z 87,A -48.4033,B 24.923,C -2.026,E1 25.1159,E2 493.3499} C_DIS
LIN {X 65.563,Y -59.1712,Z 87,A -46.6055,B 24.9235,C -2.0195,E1 25.1193,E2 491.5753} C_DIS
LIN {X 69.0614,Y -55.0479,Z 87,A -43.0228,B 24.9226,C -2.0312,E1 25.1257,E2 487.9814} C_DIS
LIN {X 71.0857,Y -52.4073,Z 87,A -40.6876,B 24.9217,C -2.0432,E1 25.1297,E2 485.6289} C_DIS
Enddeposition()
END
